LIN {X 0,Y 240.365,Z 392.146,A -85,B 0,C 180,E1 -19575.841,E2 -19575.841} C_VEL
LIN {X 0,Y 237.753,Z 387.976,A -85,B 0,C 180,E1 -19576.695,E2 -19576.695} C_VEL
LIN {X 0,Y 237.227,Z 386.044,A -85,B 0,C 180,E1 -19576.943,E2 -19576.943} C_VEL
LIN {X 0,Y 236.786,Z 383.152,A -85,B 0,C 180,E1 -19580.508,E2 -19580.508} C_VEL
LIN {X 0,Y 236.424,Z 380.849,A -85,B 0,C 180,E1 -19583.522,E2 -19583.522} C_VEL
LIN {X 0,Y 235.914,Z 377.933,A -85,B 0,C 180,E1 -19587.573,E2 -19587.573} C_VEL
LIN {X 0,Y 235.569,Z 375.427,A -85,B 0,C 180,E1 -19591.488,E2 -19591.488} C_VEL
LIN {X 0,Y 235.207,Z 373.215,A -85,B 0,C 180,E1 -19595.272,E2 -19595.272} C_VEL
LIN {X 0,Y 234.997,Z 371.839,A -85,B 0,C 180,E1 -19597.991,E2 -19597.991} C_VEL
LIN {X 0,Y 235.1,Z 371.828,A -85,B 0,C 180,E1 -19603.06,E2 -19603.06} C_VEL
LIN {X 0,Y 235.15,Z 371.825,A -85,B 0,C 180,E1 -19607.924,E2 -19607.924} C_VEL
LIN {X 0,Y 235.394,Z 371.792,A -85,B 0,C 180,E1 -19611.415,E2 -19611.415} C_VEL
LIN {X 0,Y 235.41,Z 371.786,A -85,B 0,C 180,E1 -19613.142,E2 -19613.142} C_VEL
LIN {X 0,Y 235.6,Z 371.764,A -85,B 0,C 180,E1 -19618.291,E2 -19618.291} C_VEL
LIN {X 0,Y 235.6,Z 371.763,A -85,B 0,C 180,E1 -19621.71,E2 -19621.71} C_VEL
LIN {X 0,Y 235.41,Z 371.779,A -85,B 0,C 180,E1 -19626.859,E2 -19626.859} C_VEL
LIN {X 0,Y 235.257,Z 371.795,A -85,B 0,C 180,E1 -19630.326,E2 -19630.326} C_VEL
LIN {X 0,Y 235.117,Z 371.816,A -85,B 0,C 180,E1 -19635.606,E2 -19635.606} C_VEL
LIN {X 0,Y 235.011,Z 371.808,A -85,B 0,C 180,E1 -19639.206,E2 -19639.206} C_VEL
LIN {X 0,Y 234.956,Z 371.835,A -85,B 0,C 180,E1 -19642.884,E2 -19642.884} C_VEL
LIN {X 0,Y 234.97,Z 371.815,A -85,B 0,C 180,E1 -19646.657,E2 -19646.657} C_VEL
LIN {X 0,Y 234.926,Z 371.847,A -85,B 0,C 180,E1 -19650.569,E2 -19650.569} C_VEL
LIN {X 0,Y 234.964,Z 371.826,A -85,B 0,C 180,E1 -19654.633,E2 -19654.633} C_VEL
LIN {X 0,Y 234.945,Z 371.844,A -85,B 0,C 180,E1 -19658.944,E2 -19658.944} C_VEL
LIN {X 0,Y 234.877,Z 371.898,A -85,B 0,C 180,E1 -19662.586,E2 -19662.586} C_VEL
LIN {X 0,Y 235.767,Z 374.534,A -85,B 0,C 180,E1 -19662.962,E2 -19662.962} C_VEL
LIN {X 0,Y 237.695,Z 376.657,A -85,B 0,C 180,E1 -19663.576,E2 -19663.576} C_VEL
LIN {X 0,Y 240.331,Z 380.728,A -85,B 0,C 180,E1 -19664.475,E2 -19664.475} C_VEL
LIN {X 0,Y 244.031,Z 386.932,A -85,B 0,C 180,E1 -19665.775,E2 -19665.775} C_VEL
LIN {X 0,Y 247.642,Z 393.701,A -85,B 0,C 180,E1 -19667.125,E2 -19667.125} C_VEL
LIN {X 0,Y 252.641,Z 405.359,A -85,B 0,C 180,E1 -19669.292,E2 -19669.292} C_VEL
LIN {X 0,Y 256.805,Z 418.111,A -85,B 0,C 180,E1 -19671.571,E2 -19671.571} C_VEL
LIN {X 0,Y 259.553,Z 429.821,A -85,B 0,C 180,E1 -19673.664,E2 -19673.664} C_VEL
LIN {X 0,Y 260.589,Z 437.318,A -85,B 0,C 180,E1 -19675.014,E2 -19675.014} C_VEL
LIN {X 0,Y 257.442,Z 449.414,A -85,B 0,C 180,E1 -19676.673,E2 -19676.673} C_VEL
LIN {X 0,Y 253.705,Z 461.584,A -85,B 0,C 180,E1 -19678.707,E2 -19678.707} C_VEL
LIN {X 0,Y 250.336,Z 471.991,A -85,B 0,C 180,E1 -19680.859,E2 -19680.859} C_VEL
LIN {X 0,Y 246.821,Z 481.962,A -85,B 0,C 180,E1 -19683.354,E2 -19683.354} C_VEL
LIN {X 0,Y 243.43,Z 491.106,A -85,B 0,C 180,E1 -19686.159,E2 -19686.159} C_VEL
LIN {X 0,Y 240.902,Z 497.706,A -85,B 0,C 180,E1 -19688.612,E2 -19688.612} C_VEL
LIN {X 0,Y 238.819,Z 503.332,A -85,B 0,C 180,E1 -19691.112,E2 -19691.112} C_VEL
LIN {X 0,Y 236.494,Z 509.456,A -85,B 0,C 180,E1 -19694.486,E2 -19694.486} C_VEL
LIN {X 0,Y 234.943,Z 514.169,A -85,B 0,C 180,E1 -19697.912,E2 -19697.912} C_VEL
LIN {X 0,Y 233.837,Z 517.618,A -85,B 0,C 180,E1 -19701.356,E2 -19701.356} C_VEL
LIN {X 0,Y 233.305,Z 519.888,A -85,B 0,C 180,E1 -19704.814,E2 -19704.814} C_VEL
LIN {X 0,Y 233.028,Z 521.046,A -85,B 0,C 180,E1 -19708.271,E2 -19708.271} C_VEL
LIN {X 0,Y 233.027,Z 521.058,A -85,B 0,C 180,E1 -19711.728,E2 -19711.728} C_VEL
LIN {X 0,Y 233.304,Z 519.95,A -85,B 0,C 180,E1 -19715.184,E2 -19715.184} C_VEL
LIN {X 0,Y 233.835,Z 517.729,A -85,B 0,C 180,E1 -19718.642,E2 -19718.642} C_VEL
LIN {X 0,Y 234.904,Z 514.324,A -85,B 0,C 180,E1 -19722.088,E2 -19722.088} C_VEL
LIN {X 0,Y 236.445,Z 509.661,A -85,B 0,C 180,E1 -19725.515,E2 -19725.515} C_VEL
LIN {X 0,Y 238.775,Z 503.598,A -85,B 0,C 180,E1 -19728.89,E2 -19728.89} C_VEL
LIN {X 0,Y 241.176,Z 497.014,A -85,B 0,C 180,E1 -19731.81,E2 -19731.81} C_VEL
LIN {X 0,Y 244.227,Z 489.035,A -85,B 0,C 180,E1 -19734.661,E2 -19734.661} C_VEL
LIN {X 0,Y 247.76,Z 479.453,A -85,B 0,C 180,E1 -19737.448,E2 -19737.448} C_VEL
LIN {X 0,Y 251.105,Z 469.547,A -85,B 0,C 180,E1 -19739.814,E2 -19739.814} C_VEL
LIN {X 0,Y 254.873,Z 457.976,A -85,B 0,C 180,E1 -19742.059,E2 -19742.059} C_VEL
LIN {X 0,Y 258.281,Z 446.345,A -85,B 0,C 180,E1 -19743.904,E2 -19743.904} C_VEL
LIN {X 0,Y 260.705,Z 436.623,A -85,B 0,C 180,E1 -19745.22,E2 -19745.22} C_VEL
LIN {X 0,Y 258.709,Z 425.382,A -85,B 0,C 180,E1 -19747.255,E2 -19747.255} C_VEL
LIN {X 0,Y 255.207,Z 412.553,A -85,B 0,C 180,E1 -19749.549,E2 -19749.549} C_VEL
LIN {X 0,Y 250.965,Z 401.064,A -85,B 0,C 180,E1 -19751.64,E2 -19751.64} C_VEL
LIN {X 0,Y 245.554,Z 389.421,A -85,B 0,C 180,E1 -19753.827,E2 -19753.827} C_VEL
LIN {X 0,Y 240.349,Z 380.733,A -85,B 0,C 180,E1 -19755.678,E2 -19755.678} C_VEL
LIN {X 0,Y 238.22,Z 377.466,A -85,B 0,C 180,E1 -19756.408,E2 -19756.408} C_VEL
LIN {X 0,Y 237.051,Z 376.15,A -85,B 0,C 180,E1 -19756.778,E2 -19756.778} C_VEL
LIN {X 0,Y 235.396,Z 373.796,A -85,B 0,C 180,E1 -19757.338,E2 -19757.338} C_VEL
LIN {X 0,Y 234.883,Z 371.853,A -85,B 0,C 180,E1 -19757.607,E2 -19757.607} C_VEL
LIN {X 0,Y 234.953,Z 371.842,A -85,B 0,C 180,E1 -19761.085,E2 -19761.085} C_VEL
LIN {X 0,Y 234.959,Z 371.832,A -85,B 0,C 180,E1 -19765.367,E2 -19765.367} C_VEL
LIN {X 0,Y 234.968,Z 371.841,A -85,B 0,C 180,E1 -19770.157,E2 -19770.157} C_VEL
LIN {X 0,Y 234.992,Z 371.815,A -85,B 0,C 180,E1 -19773.793,E2 -19773.793} C_VEL
LIN {X 0,Y 235.009,Z 371.806,A -85,B 0,C 180,E1 -19778.969,E2 -19778.969} C_VEL
LIN {X 0,Y 235.095,Z 371.825,A -85,B 0,C 180,E1 -19783.059,E2 -19783.059} C_VEL
LIN {X 0,Y 235.117,Z 371.793,A -85,B 0,C 180,E1 -19787.922,E2 -19787.922} C_VEL
LIN {X 0,Y 235.389,Z 371.788,A -85,B 0,C 180,E1 -19791.414,E2 -19791.414} C_VEL
LIN {X 0,Y 235.404,Z 371.788,A -85,B 0,C 180,E1 -19793.141,E2 -19793.141} C_VEL
LIN {X 0,Y 235.595,Z 371.764,A -85,B 0,C 180,E1 -19798.29,E2 -19798.29} C_VEL
LIN {X 0,Y 235.595,Z 371.766,A -85,B 0,C 180,E1 -19801.709,E2 -19801.709} C_VEL
LIN {X 0,Y 235.404,Z 371.788,A -85,B 0,C 180,E1 -19806.858,E2 -19806.858} C_VEL
LIN {X 0,Y 235.251,Z 371.806,A -85,B 0,C 180,E1 -19810.326,E2 -19810.326} C_VEL
LIN {X 0,Y 235.112,Z 371.817,A -85,B 0,C 180,E1 -19815.606,E2 -19815.606} C_VEL
LIN {X 0,Y 235.007,Z 371.836,A -85,B 0,C 180,E1 -19819.206,E2 -19819.206} C_VEL
LIN {X 0,Y 234.991,Z 371.84,A -85,B 0,C 180,E1 -19822.01,E2 -19822.01} C_VEL
LIN {X 0,Y 235.417,Z 374.315,A -85,B 0,C 180,E1 -19826.602,E2 -19826.602} C_VEL
LIN {X 0,Y 235.77,Z 376.689,A -85,B 0,C 180,E1 -19830.447,E2 -19830.447} C_VEL
LIN {X 0,Y 236.166,Z 379.419,A -85,B 0,C 180,E1 -19834.431,E2 -19834.431} C_VEL
LIN {X 0,Y 236.671,Z 382.515,A -85,B 0,C 180,E1 -19838.62,E2 -19838.62} C_VEL
LIN {X 0,Y 237.11,Z 385.372,A -85,B 0,C 180,E1 -19842.184,E2 -19842.184} C_VEL
LIN {X 0,Y 237.201,Z 386.06,A -85,B 0,C 180,E1 -19843.01,E2 -19843.01} C_VEL
LIN {X 0,Y 238.311,Z 389.145,A -85,B 0,C 180,E1 -19843.436,E2 -19843.436} C_VEL
LIN {X 0,Y 240.316,Z 392.138,A -85,B 0,C 180,E1 -19844.08,E2 -19844.08} C_VEL
LIN {X 0,Y 242.022,Z 395.595,A -85,B 0,C 180,E1 -19844.662,E2 -19844.662} C_VEL
LIN {X 0,Y 243.385,Z 398.6,A -85,B 0,C 180,E1 -19845.16,E2 -19845.16} C_VEL
LIN {X 0,Y 244.56,Z 403.788,A -85,B 0,C 180,E1 -19845.767,E2 -19845.767} C_VEL
LIN {X 0,Y 245.066,Z 416.913,A -85,B 0,C 180,E1 -19846.969,E2 -19846.969} C_VEL
LIN {X 0,Y 245.512,Z 422.315,A -85,B 0,C 180,E1 -19847.6,E2 -19847.6} C_VEL
LIN {X 0,Y 245.845,Z 423.998,A -85,B 0,C 180,E1 -19847.847,E2 -19847.847} C_VEL
LIN {X 0,Y 248.348,Z 436.665,A -85,B 0,C 180,E1 -19849.824,E2 -19849.824} C_VEL
LIN {X 0,Y 249.673,Z 447.615,A -85,B 0,C 180,E1 -19851.571,E2 -19851.571} C_VEL
LIN {X 0,Y 250.293,Z 459.212,A -85,B 0,C 180,E1 -19853.528,E2 -19853.528} C_VEL
LIN {X 0,Y 250.148,Z 467.524,A -85,B 0,C 180,E1 -19855,E2 -19855} C_VEL
LIN {X 0,Y 246.211,Z 479.542,A -85,B 0,C 180,E1 -19856.914,E2 -19856.914} C_VEL
LIN {X 0,Y 242.5,Z 490.354,A -85,B 0,C 180,E1 -19859.042,E2 -19859.042} C_VEL
LIN {X 0,Y 238.921,Z 500.373,A -85,B 0,C 180,E1 -19861.446,E2 -19861.446} C_VEL
LIN {X 0,Y 235.371,Z 510.194,A -85,B 0,C 180,E1 -19864.345,E2 -19864.345} C_VEL
LIN {X 0,Y 232.244,Z 518.392,A -85,B 0,C 180,E1 -19867.306,E2 -19867.306} C_VEL
LIN {X 0,Y 229.865,Z 525.192,A -85,B 0,C 180,E1 -19870.348,E2 -19870.348} C_VEL
LIN {X 0,Y 227.851,Z 531.486,A -85,B 0,C 180,E1 -19873.884,E2 -19873.884} C_VEL
LIN {X 0,Y 226.472,Z 536.364,A -85,B 0,C 180,E1 -19877.455,E2 -19877.455} C_VEL
LIN {X 0,Y 225.859,Z 539.958,A -85,B 0,C 180,E1 -19881.05,E2 -19881.05} C_VEL
LIN {X 0,Y 225.762,Z 542.491,A -85,B 0,C 180,E1 -19884.979,E2 -19884.979} C_VEL
LIN {X 0,Y 225.823,Z 543.533,A -85,B 0,C 180,E1 -19888.217,E2 -19888.217} C_VEL
LIN {X 0,Y 225.879,Z 543.692,A -85,B 0,C 180,E1 -19890.001,E2 -19890.001} C_VEL
LIN {X 0,Y 225.738,Z 543.065,A -85,B 0,C 180,E1 -19893.571,E2 -19893.571} C_VEL
LIN {X 0,Y 225.79,Z 541.267,A -85,B 0,C 180,E1 -19897.153,E2 -19897.153} C_VEL
LIN {X 0,Y 226.079,Z 538.274,A -85,B 0,C 180,E1 -19900.75,E2 -19900.75} C_VEL
LIN {X 0,Y 227.108,Z 534.042,A -85,B 0,C 180,E1 -19904.334,E2 -19904.334} C_VEL
LIN {X 0,Y 228.777,Z 528.453,A -85,B 0,C 180,E1 -19907.891,E2 -19907.891} C_VEL
LIN {X 0,Y 231.143,Z 521.361,A -85,B 0,C 180,E1 -19911.4,E2 -19911.4} C_VEL
LIN {X 0,Y 233.997,Z 513.801,A -85,B 0,C 180,E1 -19914.393,E2 -19914.393} C_VEL
LIN {X 0,Y 237.628,Z 503.825,A -85,B 0,C 180,E1 -19917.576,E2 -19917.576} C_VEL
LIN {X 0,Y 241.296,Z 493.766,A -85,B 0,C 180,E1 -19920.161,E2 -19920.161} C_VEL
LIN {X 0,Y 245.546,Z 481.496,A -85,B 0,C 180,E1 -19922.701,E2 -19922.701} C_VEL
LIN {X 0,Y 249.696,Z 468.862,A -85,B 0,C 180,E1 -19924.775,E2 -19924.775} C_VEL
LIN {X 0,Y 250.205,Z 466.104,A -85,B 0,C 180,E1 -19925.212,E2 -19925.212} C_VEL
LIN {X 0,Y 250.129,Z 454.413,A -85,B 0,C 180,E1 -19927.251,E2 -19927.251} C_VEL
LIN {X 0,Y 249.121,Z 442.557,A -85,B 0,C 180,E1 -19929.202,E2 -19929.202} C_VEL
LIN {X 0,Y 247.216,Z 430.307,A -85,B 0,C 180,E1 -19931.117,E2 -19931.117} C_VEL
LIN {X 0,Y 243.831,Z 416.677,A -85,B 0,C 180,E1 -19933.258,E2 -19933.258} C_VEL
LIN {X 0,Y 239.847,Z 404.951,A -85,B 0,C 180,E1 -19935.158,E2 -19935.158} C_VEL
LIN {X 0,Y 237.479,Z 399.928,A -85,B 0,C 180,E1 -19936.083,E2 -19936.083} C_VEL
LIN {X 0,Y 235.391,Z 395.789,A -85,B 0,C 180,E1 -19936.883,E2 -19936.883} C_VEL
LIN {X 0,Y 233.368,Z 392.047,A -85,B 0,C 180,E1 -19937.617,E2 -19937.617} C_VEL
LIN {X 0,Y 232.475,Z 390.688,A -85,B 0,C 180,E1 -19937.927,E2 -19937.927} C_VEL
LIN {X 0,Y 230.569,Z 387.673,A -85,B 0,C 180,E1 -19938.61,E2 -19938.61} C_VEL
LIN {X 0,Y 229.99,Z 385.549,A -85,B 0,C 180,E1 -19938.915,E2 -19938.915} C_VEL
LIN {X 0,Y 229.487,Z 382.624,A -85,B 0,C 180,E1 -19942.774,E2 -19942.774} C_VEL
LIN {X 0,Y 229.09,Z 380.015,A -85,B 0,C 180,E1 -19946.482,E2 -19946.482} C_VEL
LIN {X 0,Y 228.665,Z 377.405,A -85,B 0,C 180,E1 -19950.544,E2 -19950.544} C_VEL
LIN {X 0,Y 228.33,Z 375.085,A -85,B 0,C 180,E1 -19954.474,E2 -19954.474} C_VEL
LIN {X 0,Y 228.007,Z 373.088,A -85,B 0,C 180,E1 -19958.292,E2 -19958.292} C_VEL
LIN {X 0,Y 228.007,Z 372.71,A -85,B 0,C 180,E1 -19962.047,E2 -19962.047} C_VEL
LIN {X 0,Y 228.069,Z 372.705,A -85,B 0,C 180,E1 -19965.728,E2 -19965.728} C_VEL
LIN {X 0,Y 228.329,Z 372.672,A -85,B 0,C 180,E1 -19971.147,E2 -19971.147} C_VEL
LIN {X 0,Y 228.362,Z 372.665,A -85,B 0,C 180,E1 -19972.929,E2 -19972.929} C_VEL
LIN {X 0,Y 228.559,Z 372.642,A -85,B 0,C 180,E1 -19978.238,E2 -19978.238} C_VEL
LIN {X 0,Y 228.559,Z 372.64,A -85,B 0,C 180,E1 -19981.762,E2 -19981.762} C_VEL
LIN {X 0,Y 228.362,Z 372.657,A -85,B 0,C 180,E1 -19987.071,E2 -19987.071} C_VEL
LIN {X 0,Y 228.171,Z 372.67,A -85,B 0,C 180,E1 -19990.65,E2 -19990.65} C_VEL
LIN {X 0,Y 228.068,Z 372.671,A -85,B 0,C 180,E1 -19994.272,E2 -19994.272} C_VEL
LIN {X 0,Y 228.006,Z 372.699,A -85,B 0,C 180,E1 -19997.953,E2 -19997.953} C_VEL
LIN {X 0,Y 227.92,Z 372.7,A -85,B 0,C 180,E1 -20002.321,E2 -20002.321} C_VEL
LIN {X 0,Y 227.945,Z 372.689,A -85,B 0,C 180,E1 -20006.602,E2 -20006.602} C_VEL
LIN {X 0,Y 227.901,Z 372.722,A -85,B 0,C 180,E1 -20010.291,E2 -20010.291} C_VEL
LIN {X 0,Y 227.893,Z 372.7,A -85,B 0,C 180,E1 -20013.718,E2 -20013.718} C_VEL
LIN {X 0,Y 227.873,Z 372.726,A -85,B 0,C 180,E1 -20018.086,E2 -20018.086} C_VEL
LIN {X 0,Y 227.84,Z 372.737,A -85,B 0,C 180,E1 -20020.64,E2 -20020.64} C_VEL
LIN {X 0,Y 228.705,Z 375.293,A -85,B 0,C 180,E1 -20021.039,E2 -20021.039} C_VEL
LIN {X 0,Y 230.755,Z 377.617,A -85,B 0,C 180,E1 -20021.757,E2 -20021.757} C_VEL
LIN {X 0,Y 233.487,Z 381.79,A -85,B 0,C 180,E1 -20022.776,E2 -20022.776} C_VEL
LIN {X 0,Y 234.607,Z 383.303,A -85,B 0,C 180,E1 -20023.182,E2 -20023.182} C_VEL
LIN {X 0,Y 237.64,Z 388.184,A -85,B 0,C 180,E1 -20024.322,E2 -20024.322} C_VEL
LIN {X 0,Y 242.189,Z 396.617,A -85,B 0,C 180,E1 -20026.156,E2 -20026.156} C_VEL
LIN {X 0,Y 246.882,Z 407.826,A -85,B 0,C 180,E1 -20028.354,E2 -20028.354} C_VEL
LIN {X 0,Y 250.522,Z 419.001,A -85,B 0,C 180,E1 -20030.486,E2 -20030.486} C_VEL
LIN {X 0,Y 253.168,Z 430.055,A -85,B 0,C 180,E1 -20032.567,E2 -20032.567} C_VEL
LIN {X 0,Y 254.483,Z 438.888,A -85,B 0,C 180,E1 -20034.255,E2 -20034.255} C_VEL
LIN {X 0,Y 251.197,Z 450.93,A -85,B 0,C 180,E1 -20035.974,E2 -20035.974} C_VEL
LIN {X 0,Y 247.655,Z 461.936,A -85,B 0,C 180,E1 -20037.852,E2 -20037.852} C_VEL
LIN {X 0,Y 244.059,Z 472.582,A -85,B 0,C 180,E1 -20040.099,E2 -20040.099} C_VEL
LIN {X 0,Y 240.456,Z 482.315,A -85,B 0,C 180,E1 -20042.59,E2 -20042.59} C_VEL
LIN {X 0,Y 236.933,Z 491.457,A -85,B 0,C 180,E1 -20045.463,E2 -20045.463} C_VEL
LIN {X 0,Y 234.286,Z 498.057,A -85,B 0,C 180,E1 -20047.977,E2 -20047.977} C_VEL
LIN {X 0,Y 232.082,Z 503.683,A -85,B 0,C 180,E1 -20050.542,E2 -20050.542} C_VEL
LIN {X 0,Y 230.228,Z 508.403,A -85,B 0,C 180,E1 -20053.141,E2 -20053.141} C_VEL
LIN {X 0,Y 228.342,Z 513.477,A -85,B 0,C 180,E1 -20056.653,E2 -20056.653} C_VEL
LIN {X 0,Y 227.331,Z 516.395,A -85,B 0,C 180,E1 -20059.309,E2 -20059.309} C_VEL
LIN {X 0,Y 226.382,Z 519.591,A -85,B 0,C 180,E1 -20063.433,E2 -20063.433} C_VEL
LIN {X 0,Y 226.111,Z 520.949,A -85,B 0,C 180,E1 -20066.435,E2 -20066.435} C_VEL
LIN {X 0,Y 225.919,Z 521.547,A -85,B 0,C 180,E1 -20069.999,E2 -20069.999} C_VEL
LIN {X 0,Y 226.088,Z 520.987,A -85,B 0,C 180,E1 -20073.564,E2 -20073.564} C_VEL
LIN {X 0,Y 226.491,Z 519.329,A -85,B 0,C 180,E1 -20077.129,E2 -20077.129} C_VEL
LIN {X 0,Y 227.318,Z 516.526,A -85,B 0,C 180,E1 -20080.69,E2 -20080.69} C_VEL
LIN {X 0,Y 228.716,Z 512.504,A -85,B 0,C 180,E1 -20084.23,E2 -20084.23} C_VEL
LIN {X 0,Y 230.799,Z 507.158,A -85,B 0,C 180,E1 -20087.728,E2 -20087.728} C_VEL
LIN {X 0,Y 233.367,Z 500.345,A -85,B 0,C 180,E1 -20091.185,E2 -20091.185} C_VEL
LIN {X 0,Y 236.849,Z 491.814,A -85,B 0,C 180,E1 -20094.545,E2 -20094.545} C_VEL
LIN {X 0,Y 240.344,Z 482.74,A -85,B 0,C 180,E1 -20097.422,E2 -20097.422} C_VEL
LIN {X 0,Y 243.753,Z 473.62,A -85,B 0,C 180,E1 -20099.785,E2 -20099.785} C_VEL
LIN {X 0,Y 247.51,Z 462.49,A -85,B 0,C 180,E1 -20102.167,E2 -20102.167} C_VEL
LIN {X 0,Y 251.417,Z 450.423,A -85,B 0,C 180,E1 -20104.232,E2 -20104.232} C_VEL
LIN {X 0,Y 254.499,Z 439.294,A -85,B 0,C 180,E1 -20105.809,E2 -20105.809} C_VEL
LIN {X 0,Y 253.158,Z 429.641,A -85,B 0,C 180,E1 -20107.643,E2 -20107.643} C_VEL
LIN {X 0,Y 250.331,Z 418.167,A -85,B 0,C 180,E1 -20109.808,E2 -20109.808} C_VEL
LIN {X 0,Y 246.696,Z 407.16,A -85,B 0,C 180,E1 -20111.904,E2 -20111.904} C_VEL
LIN {X 0,Y 241.928,Z 395.995,A -85,B 0,C 180,E1 -20114.117,E2 -20114.117} C_VEL
LIN {X 0,Y 237.89,Z 388.617,A -85,B 0,C 180,E1 -20115.737,E2 -20115.737} C_VEL
LIN {X 0,Y 236.099,Z 385.655,A -85,B 0,C 180,E1 -20116.425,E2 -20116.425} C_VEL
LIN {X 0,Y 233.646,Z 381.958,A -85,B 0,C 180,E1 -20117.333,E2 -20117.333} C_VEL
LIN {X 0,Y 231.567,Z 378.932,A -85,B 0,C 180,E1 -20118.11,E2 -20118.11} C_VEL
LIN {X 0,Y 230.784,Z 377.645,A -85,B 0,C 180,E1 -20118.401,E2 -20118.401} C_VEL
LIN {X 0,Y 228.634,Z 375.23,A -85,B 0,C 180,E1 -20119.157,E2 -20119.157} C_VEL
LIN {X 0,Y 227.853,Z 372.728,A -85,B 0,C 180,E1 -20119.575,E2 -20119.575} C_VEL
LIN {X 0,Y 227.899,Z 372.724,A -85,B 0,C 180,E1 -20124.131,E2 -20124.131} C_VEL
LIN {X 0,Y 227.871,Z 372.712,A -85,B 0,C 180,E1 -20128.378,E2 -20128.378} C_VEL
LIN {X 0,Y 227.884,Z 372.698,A -85,B 0,C 180,E1 -20132.445,E2 -20132.445} C_VEL
LIN {X 0,Y 227.913,Z 372.719,A -85,B 0,C 180,E1 -20136.367,E2 -20136.367} C_VEL
LIN {X 0,Y 227.941,Z 372.686,A -85,B 0,C 180,E1 -20140.174,E2 -20140.174} C_VEL
LIN {X 0,Y 228.056,Z 372.7,A -85,B 0,C 180,E1 -20143.898,E2 -20143.898} C_VEL
LIN {X 0,Y 228.074,Z 372.667,A -85,B 0,C 180,E1 -20147.543,E2 -20147.543} C_VEL
LIN {X 0,Y 228.323,Z 372.669,A -85,B 0,C 180,E1 -20151.147,E2 -20151.147} C_VEL
LIN {X 0,Y 228.357,Z 372.667,A -85,B 0,C 180,E1 -20152.928,E2 -20152.928} C_VEL
LIN {X 0,Y 228.553,Z 372.641,A -85,B 0,C 180,E1 -20158.238,E2 -20158.238} C_VEL
LIN {X 0,Y 228.554,Z 372.643,A -85,B 0,C 180,E1 -20161.762,E2 -20161.762} C_VEL
LIN {X 0,Y 228.356,Z 372.667,A -85,B 0,C 180,E1 -20167.071,E2 -20167.071} C_VEL
LIN {X 0,Y 228.165,Z 372.69,A -85,B 0,C 180,E1 -20170.65,E2 -20170.65} C_VEL
LIN {X 0,Y 228.063,Z 372.701,A -85,B 0,C 180,E1 -20174.272,E2 -20174.272} C_VEL
LIN {X 0,Y 228.001,Z 372.705,A -85,B 0,C 180,E1 -20177.953,E2 -20177.953} C_VEL
LIN {X 0,Y 227.94,Z 372.717,A -85,B 0,C 180,E1 -20179.825,E2 -20179.825} C_VEL
LIN {X 0,Y 228.07,Z 373.495,A -85,B 0,C 180,E1 -20182.416,E2 -20182.416} C_VEL
LIN {X 0,Y 228.466,Z 375.895,A -85,B 0,C 180,E1 -20186.865,E2 -20186.865} C_VEL
LIN {X 0,Y 228.85,Z 378.715,A -85,B 0,C 180,E1 -20191.471,E2 -20191.471} C_VEL
LIN {X 0,Y 229.289,Z 381.526,A -85,B 0,C 180,E1 -20195.617,E2 -20195.617} C_VEL
LIN {X 0,Y 229.933,Z 385.158,A -85,B 0,C 180,E1 -20200.53,E2 -20200.53} C_VEL
LIN {X 0,Y 229.974,Z 385.548,A -85,B 0,C 180,E1 -20201.019,E2 -20201.019} C_VEL
LIN {X 0,Y 231.049,Z 388.684,A -85,B 0,C 180,E1 -20201.501,E2 -20201.501} C_VEL
LIN {X 0,Y 233.27,Z 391.819,A -85,B 0,C 180,E1 -20202.272,E2 -20202.272} C_VEL
LIN {X 0,Y 235.336,Z 395.727,A -85,B 0,C 180,E1 -20203.028,E2 -20203.028} C_VEL
LIN {X 0,Y 236.747,Z 398.488,A -85,B 0,C 180,E1 -20203.572,E2 -20203.572} C_VEL
LIN {X 0,Y 239.144,Z 403.362,A -85,B 0,C 180,E1 -20204.485,E2 -20204.485} C_VEL
LIN {X 0,Y 241.953,Z 410.536,A -85,B 0,C 180,E1 -20205.708,E2 -20205.708} C_VEL
LIN {X 0,Y 245.208,Z 421.548,A -85,B 0,C 180,E1 -20207.458,E2 -20207.458} C_VEL
LIN {X 0,Y 245.845,Z 423.998,A -85,B 0,C 180,E1 -20207.847,E2 -20207.847} C_VEL
LIN {X 0,Y 246.467,Z 429.079,A -85,B 0,C 180,E1 -20208.532,E2 -20208.532} C_VEL
LIN {X 0,Y 246.138,Z 434.527,A -85,B 0,C 180,E1 -20209.122,E2 -20209.122} C_VEL
LIN {X 0,Y 244.334,Z 445.278,A -85,B 0,C 180,E1 -20210.273,E2 -20210.273} C_VEL
LIN {X 0,Y 243.794,Z 450.476,A -85,B 0,C 180,E1 -20210.973,E2 -20210.973} C_VEL
LIN {X 0,Y 243.798,Z 452.076,A -85,B 0,C 180,E1 -20211.239,E2 -20211.239} C_VEL
LIN {X 0,Y 244.081,Z 463.437,A -85,B 0,C 180,E1 -20213.275,E2 -20213.275} C_VEL
LIN {X 0,Y 243.907,Z 468.567,A -85,B 0,C 180,E1 -20214.24,E2 -20214.24} C_VEL
LIN {X 0,Y 239.54,Z 481.348,A -85,B 0,C 180,E1 -20216.374,E2 -20216.374} C_VEL
LIN {X 0,Y 235.086,Z 493.575,A -85,B 0,C 180,E1 -20218.957,E2 -20218.957} C_VEL
LIN {X 0,Y 231.044,Z 504.241,A -85,B 0,C 180,E1 -20221.787,E2 -20221.787} C_VEL
LIN {X 0,Y 227.513,Z 513.563,A -85,B 0,C 180,E1 -20224.866,E2 -20224.866} C_VEL
LIN {X 0,Y 224.458,Z 521.11,A -85,B 0,C 180,E1 -20227.931,E2 -20227.931} C_VEL
LIN {X 0,Y 221.94,Z 528.174,A -85,B 0,C 180,E1 -20231.54,E2 -20231.54} C_VEL
LIN {X 0,Y 220.135,Z 533.742,A -85,B 0,C 180,E1 -20235.203,E2 -20235.203} C_VEL
LIN {X 0,Y 219.058,Z 537.967,A -85,B 0,C 180,E1 -20238.902,E2 -20238.902} C_VEL
LIN {X 0,Y 218.625,Z 540.943,A -85,B 0,C 180,E1 -20242.613,E2 -20242.613} C_VEL
LIN {X 0,Y 218.641,Z 542.729,A -85,B 0,C 180,E1 -20246.315,E2 -20246.315} C_VEL
LIN {X 0,Y 218.81,Z 543.346,A -85,B 0,C 180,E1 -20250.001,E2 -20250.001} C_VEL
LIN {X 0,Y 218.647,Z 542.716,A -85,B 0,C 180,E1 -20253.687,E2 -20253.687} C_VEL
LIN {X 0,Y 218.69,Z 540.916,A -85,B 0,C 180,E1 -20257.386,E2 -20257.386} C_VEL
LIN {X 0,Y 219.059,Z 537.923,A -85,B 0,C 180,E1 -20261.099,E2 -20261.099} C_VEL
LIN {X 0,Y 220.152,Z 533.689,A -85,B 0,C 180,E1 -20264.797,E2 -20264.797} C_VEL
LIN {X 0,Y 221.941,Z 528.099,A -85,B 0,C 180,E1 -20268.462,E2 -20268.462} C_VEL
LIN {X 0,Y 224.458,Z 521.007,A -85,B 0,C 180,E1 -20272.07,E2 -20272.07} C_VEL
LIN {X 0,Y 227.486,Z 513.448,A -85,B 0,C 180,E1 -20275.138,E2 -20275.138} C_VEL
LIN {X 0,Y 231.164,Z 503.815,A -85,B 0,C 180,E1 -20278.3,E2 -20278.3} C_VEL
LIN {X 0,Y 235.133,Z 493.413,A -85,B 0,C 180,E1 -20281.038,E2 -20281.038} C_VEL
LIN {X 0,Y 239.544,Z 481.142,A -85,B 0,C 180,E1 -20283.627,E2 -20283.627} C_VEL
LIN {X 0,Y 243.856,Z 468.502,A -85,B 0,C 180,E1 -20285.734,E2 -20285.734} C_VEL
LIN {X 0,Y 243.999,Z 455.668,A -85,B 0,C 180,E1 -20288.086,E2 -20288.086} C_VEL
LIN {X 0,Y 242.91,Z 441.93,A -85,B 0,C 180,E1 -20290.442,E2 -20290.442} C_VEL
LIN {X 0,Y 241.157,Z 430.791,A -85,B 0,C 180,E1 -20292.276,E2 -20292.276} C_VEL
LIN {X 0,Y 237.893,Z 417.634,A -85,B 0,C 180,E1 -20294.488,E2 -20294.488} C_VEL
LIN {X 0,Y 234.926,Z 408.704,A -85,B 0,C 180,E1 -20296.035,E2 -20296.035} C_VEL
LIN {X 0,Y 231.654,Z 401.363,A -85,B 0,C 180,E1 -20297.47,E2 -20297.47} C_VEL
LIN {X 0,Y 228.463,Z 395.691,A -85,B 0,C 180,E1 -20298.741,E2 -20298.741} C_VEL
LIN {X 0,Y 226.406,Z 392,A -85,B 0,C 180,E1 -20299.557,E2 -20299.557} C_VEL
LIN {X 0,Y 225.713,Z 390.621,A -85,B 0,C 180,E1 -20299.839,E2 -20299.839} C_VEL
LIN {X 0,Y 223.485,Z 387.605,A -85,B 0,C 180,E1 -20300.686,E2 -20300.686} C_VEL
LIN {X 0,Y 222.657,Z 385.012,A -85,B 0,C 180,E1 -20301.136,E2 -20301.136} C_VEL
LIN {X 0,Y 222.195,Z 382.085,A -85,B 0,C 180,E1 -20305.325,E2 -20305.325} C_VEL
LIN {X 0,Y 221.774,Z 379.363,A -85,B 0,C 180,E1 -20309.534,E2 -20309.534} C_VEL
LIN {X 0,Y 221.45,Z 376.969,A -85,B 0,C 180,E1 -20313.621,E2 -20313.621} C_VEL
LIN {X 0,Y 221.098,Z 374.921,A -85,B 0,C 180,E1 -20317.577,E2 -20317.577} C_VEL
LIN {X 0,Y 220.935,Z 373.999,A -85,B 0,C 180,E1 -20319.518,E2 -20319.518} C_VEL
LIN {X 0,Y 220.988,Z 373.586,A -85,B 0,C 180,E1 -20322.571,E2 -20322.571} C_VEL
LIN {X 0,Y 221.03,Z 373.583,A -85,B 0,C 180,E1 -20327.14,E2 -20327.14} C_VEL
LIN {X 0,Y 221.262,Z 373.554,A -85,B 0,C 180,E1 -20330.862,E2 -20330.862} C_VEL
LIN {X 0,Y 221.315,Z 373.545,A -85,B 0,C 180,E1 -20332.703,E2 -20332.703} C_VEL
LIN {X 0,Y 221.517,Z 373.519,A -85,B 0,C 180,E1 -20338.182,E2 -20338.182} C_VEL
LIN {X 0,Y 221.517,Z 373.517,A -85,B 0,C 180,E1 -20341.818,E2 -20341.818} C_VEL
LIN {X 0,Y 221.315,Z 373.535,A -85,B 0,C 180,E1 -20347.298,E2 -20347.298} C_VEL
LIN {X 0,Y 221.115,Z 373.541,A -85,B 0,C 180,E1 -20350.994,E2 -20350.994} C_VEL
LIN {X 0,Y 221.02,Z 373.579,A -85,B 0,C 180,E1 -20356.63,E2 -20356.63} C_VEL
LIN {X 0,Y 220.888,Z 373.559,A -85,B 0,C 180,E1 -20360.487,E2 -20360.487} C_VEL
LIN {X 0,Y 220.866,Z 373.596,A -85,B 0,C 180,E1 -20364.435,E2 -20364.435} C_VEL
LIN {X 0,Y 220.83,Z 373.579,A -85,B 0,C 180,E1 -20368.515,E2 -20368.515} C_VEL
LIN {X 0,Y 220.826,Z 373.581,A -85,B 0,C 180,E1 -20372.755,E2 -20372.755} C_VEL
LIN {X 0,Y 220.842,Z 373.602,A -85,B 0,C 180,E1 -20377.288,E2 -20377.288} C_VEL
LIN {X 0,Y 220.847,Z 373.684,A -85,B 0,C 180,E1 -20378.501,E2 -20378.501} C_VEL
LIN {X 0,Y 221.651,Z 376.192,A -85,B 0,C 180,E1 -20378.918,E2 -20378.918} C_VEL
LIN {X 0,Y 223.631,Z 378.416,A -85,B 0,C 180,E1 -20379.683,E2 -20379.683} C_VEL
LIN {X 0,Y 224.483,Z 379.429,A -85,B 0,C 180,E1 -20380.008,E2 -20380.008} C_VEL
LIN {X 0,Y 226.542,Z 382.669,A -85,B 0,C 180,E1 -20380.868,E2 -20380.868} C_VEL
LIN {X 0,Y 227.861,Z 384.392,A -85,B 0,C 180,E1 -20381.386,E2 -20381.386} C_VEL
LIN {X 0,Y 231.25,Z 389.629,A -85,B 0,C 180,E1 -20382.763,E2 -20382.763} C_VEL
LIN {X 0,Y 234.891,Z 395.831,A -85,B 0,C 180,E1 -20384.288,E2 -20384.288} C_VEL
LIN {X 0,Y 239.012,Z 404.711,A -85,B 0,C 180,E1 -20386.239,E2 -20386.239} C_VEL
LIN {X 0,Y 243.335,Z 416.6,A -85,B 0,C 180,E1 -20388.671,E2 -20388.671} C_VEL
LIN {X 0,Y 246.184,Z 427.476,A -85,B 0,C 180,E1 -20390.844,E2 -20390.844} C_VEL
LIN {X 0,Y 248.118,Z 438.211,A -85,B 0,C 180,E1 -20392.996,E2 -20392.996} C_VEL
LIN {X 0,Y 248.271,Z 440.971,A -85,B 0,C 180,E1 -20393.525,E2 -20393.525} C_VEL
LIN {X 0,Y 244.601,Z 453.612,A -85,B 0,C 180,E1 -20395.425,E2 -20395.425} C_VEL
LIN {X 0,Y 240.989,Z 464.223,A -85,B 0,C 180,E1 -20397.348,E2 -20397.348} C_VEL
LIN {X 0,Y 237.755,Z 473.397,A -85,B 0,C 180,E1 -20399.352,E2 -20399.352} C_VEL
LIN {X 0,Y 233.638,Z 484.104,A -85,B 0,C 180,E1 -20402.208,E2 -20402.208} C_VEL
LIN {X 0,Y 229.99,Z 493.017,A -85,B 0,C 180,E1 -20405.154,E2 -20405.154} C_VEL
LIN {X 0,Y 226.491,Z 501.284,A -85,B 0,C 180,E1 -20408.576,E2 -20408.576} C_VEL
LIN {X 0,Y 224.099,Z 507.275,A -85,B 0,C 180,E1 -20411.722,E2 -20411.722} C_VEL
LIN {X 0,Y 221.867,Z 512.678,A -85,B 0,C 180,E1 -20415.32,E2 -20415.32} C_VEL
LIN {X 0,Y 220.345,Z 516.744,A -85,B 0,C 180,E1 -20418.966,E2 -20418.966} C_VEL
LIN {X 0,Y 219.435,Z 519.592,A -85,B 0,C 180,E1 -20422.639,E2 -20422.639} C_VEL
LIN {X 0,Y 219.031,Z 521.297,A -85,B 0,C 180,E1 -20426.32,E2 -20426.32} C_VEL
LIN {X 0,Y 218.85,Z 521.894,A -85,B 0,C 180,E1 -20429.999,E2 -20429.999} C_VEL
LIN {X 0,Y 219.009,Z 521.334,A -85,B 0,C 180,E1 -20433.679,E2 -20433.679} C_VEL
LIN {X 0,Y 219.434,Z 519.677,A -85,B 0,C 180,E1 -20437.36,E2 -20437.36} C_VEL
LIN {X 0,Y 220.33,Z 516.874,A -85,B 0,C 180,E1 -20441.033,E2 -20441.033} C_VEL
LIN {X 0,Y 221.811,Z 512.852,A -85,B 0,C 180,E1 -20444.683,E2 -20444.683} C_VEL
LIN {X 0,Y 224.012,Z 507.506,A -85,B 0,C 180,E1 -20448.283,E2 -20448.283} C_VEL
LIN {X 0,Y 226.74,Z 500.692,A -85,B 0,C 180,E1 -20451.835,E2 -20451.835} C_VEL
LIN {X 0,Y 230.386,Z 492.161,A -85,B 0,C 180,E1 -20455.281,E2 -20455.281} C_VEL
LIN {X 0,Y 234.057,Z 483.086,A -85,B 0,C 180,E1 -20458.223,E2 -20458.223} C_VEL
LIN {X 0,Y 237.988,Z 472.859,A -85,B 0,C 180,E1 -20460.906,E2 -20460.906} C_VEL
LIN {X 0,Y 241.886,Z 461.847,A -85,B 0,C 180,E1 -20463.257,E2 -20463.257} C_VEL
LIN {X 0,Y 245.915,Z 449.588,A -85,B 0,C 180,E1 -20465.36,E2 -20465.36} C_VEL
LIN {X 0,Y 248.428,Z 440.948,A -85,B 0,C 180,E1 -20466.592,E2 -20466.592} C_VEL
LIN {X 0,Y 246.83,Z 430.03,A -85,B 0,C 180,E1 -20468.785,E2 -20468.785} C_VEL
LIN {X 0,Y 243.968,Z 418.528,A -85,B 0,C 180,E1 -20471.071,E2 -20471.071} C_VEL
LIN {X 0,Y 239.982,Z 406.96,A -85,B 0,C 180,E1 -20473.431,E2 -20473.431} C_VEL
LIN {X 0,Y 236.044,Z 398.094,A -85,B 0,C 180,E1 -20475.347,E2 -20475.347} C_VEL
LIN {X 0,Y 232.097,Z 390.945,A -85,B 0,C 180,E1 -20477.054,E2 -20477.054} C_VEL
LIN {X 0,Y 229.558,Z 387.025,A -85,B 0,C 180,E1 -20478.103,E2 -20478.103} C_VEL
LIN {X 0,Y 226.842,Z 382.97,A -85,B 0,C 180,E1 -20479.192,E2 -20479.192} C_VEL
LIN {X 0,Y 224.751,Z 380.006,A -85,B 0,C 180,E1 -20480.05,E2 -20480.05} C_VEL
LIN {X 0,Y 223.941,Z 378.656,A -85,B 0,C 180,E1 -20480.383,E2 -20480.383} C_VEL
LIN {X 0,Y 221.819,Z 376.486,A -85,B 0,C 180,E1 -20481.19,E2 -20481.19} C_VEL
LIN {X 0,Y 220.885,Z 373.95,A -85,B 0,C 180,E1 -20481.653,E2 -20481.653} C_VEL
LIN {X 0,Y 220.841,Z 373.601,A -85,B 0,C 180,E1 -20481.789,E2 -20481.789} C_VEL
LIN {X 0,Y 220.819,Z 373.587,A -85,B 0,C 180,E1 -20485.841,E2 -20485.841} C_VEL
LIN {X 0,Y 220.867,Z 373.598,A -85,B 0,C 180,E1 -20489.394,E2 -20489.394} C_VEL
LIN {X 0,Y 220.894,Z 373.569,A -85,B 0,C 180,E1 -20493.549,E2 -20493.549} C_VEL
LIN {X 0,Y 220.876,Z 373.581,A -85,B 0,C 180,E1 -20497.553,E2 -20497.553} C_VEL
LIN {X 0,Y 220.983,Z 373.581,A -85,B 0,C 180,E1 -20502.571,E2 -20502.571} C_VEL
LIN {X 0,Y 221.012,Z 373.544,A -85,B 0,C 180,E1 -20507.138,E2 -20507.138} C_VEL
LIN {X 0,Y 221.257,Z 373.551,A -85,B 0,C 180,E1 -20510.861,E2 -20510.861} C_VEL
LIN {X 0,Y 221.31,Z 373.544,A -85,B 0,C 180,E1 -20512.702,E2 -20512.702} C_VEL
LIN {X 0,Y 221.511,Z 373.518,A -85,B 0,C 180,E1 -20518.182,E2 -20518.182} C_VEL
LIN {X 0,Y 221.512,Z 373.52,A -85,B 0,C 180,E1 -20521.818,E2 -20521.818} C_VEL
LIN {X 0,Y 221.309,Z 373.545,A -85,B 0,C 180,E1 -20527.298,E2 -20527.298} C_VEL
LIN {X 0,Y 221.109,Z 373.569,A -85,B 0,C 180,E1 -20530.994,E2 -20530.994} C_VEL
LIN {X 0,Y 221.014,Z 373.577,A -85,B 0,C 180,E1 -20536.63,E2 -20536.63} C_VEL
LIN {X 0,Y 220.92,Z 373.586,A -85,B 0,C 180,E1 -20538.549,E2 -20538.549} C_VEL
LIN {X 0,Y 220.938,Z 374.054,A -85,B 0,C 180,E1 -20540.481,E2 -20540.481} C_VEL
LIN {X 0,Y 221.242,Z 375.965,A -85,B 0,C 180,E1 -20544.391,E2 -20544.391} C_VEL
LIN {X 0,Y 221.594,Z 378.19,A -85,B 0,C 180,E1 -20548.407,E2 -20548.407} C_VEL
LIN {X 0,Y 221.979,Z 380.731,A -85,B 0,C 180,E1 -20552.563,E2 -20552.563} C_VEL
LIN {X 0,Y 222.447,Z 383.653,A -85,B 0,C 180,E1 -20556.89,E2 -20556.89} C_VEL
LIN {X 0,Y 222.641,Z 385.031,A -85,B 0,C 180,E1 -20558.821,E2 -20558.821} C_VEL
LIN {X 0,Y 223.863,Z 388.314,A -85,B 0,C 180,E1 -20559.385,E2 -20559.385} C_VEL
LIN {X 0,Y 226.253,Z 391.564,A -85,B 0,C 180,E1 -20560.292,E2 -20560.292} C_VEL
LIN {X 0,Y 228.231,Z 395.342,A -85,B 0,C 180,E1 -20561.09,E2 -20561.09} C_VEL
LIN {X 0,Y 229.534,Z 397.48,A -85,B 0,C 180,E1 -20561.608,E2 -20561.608} C_VEL
LIN {X 0,Y 232.985,Z 404.32,A -85,B 0,C 180,E1 -20563.038,E2 -20563.038} C_VEL
LIN {X 0,Y 235.741,Z 410.712,A -85,B 0,C 180,E1 -20564.268,E2 -20564.268} C_VEL
LIN {X 0,Y 238.895,Z 420.805,A -85,B 0,C 180,E1 -20566.016,E2 -20566.016} C_VEL
LIN {X 0,Y 241.739,Z 433.58,A -85,B 0,C 180,E1 -20568.127,E2 -20568.127} C_VEL
LIN {X 0,Y 243.382,Z 445.516,A -85,B 0,C 180,E1 -20570.131,E2 -20570.131} C_VEL
LIN {X 0,Y 243.798,Z 452.076,A -85,B 0,C 180,E1 -20571.239,E2 -20571.239} C_VEL
LIN {X 0,Y 243.333,Z 457.097,A -85,B 0,C 180,E1 -20572.001,E2 -20572.001} C_VEL
LIN {X 0,Y 241.88,Z 462.132,A -85,B 0,C 180,E1 -20572.659,E2 -20572.659} C_VEL
LIN {X 0,Y 237.408,Z 472.066,A -85,B 0,C 180,E1 -20573.94,E2 -20573.94} C_VEL
LIN {X 0,Y 234.584,Z 478.43,A -85,B 0,C 180,E1 -20574.94,E2 -20574.94} C_VEL
LIN {X 0,Y 230.348,Z 489.659,A -85,B 0,C 180,E1 -20577.211,E2 -20577.211} C_VEL
LIN {X 0,Y 226.404,Z 499.674,A -85,B 0,C 180,E1 -20579.707,E2 -20579.707} C_VEL
LIN {X 0,Y 222.464,Z 509.491,A -85,B 0,C 180,E1 -20582.738,E2 -20582.738} C_VEL
LIN {X 0,Y 219.095,Z 517.693,A -85,B 0,C 180,E1 -20585.86,E2 -20585.86} C_VEL
LIN {X 0,Y 216.372,Z 524.49,A -85,B 0,C 180,E1 -20589.067,E2 -20589.067} C_VEL
LIN {X 0,Y 214.069,Z 530.783,A -85,B 0,C 180,E1 -20592.815,E2 -20592.815} C_VEL
LIN {X 0,Y 212.526,Z 535.664,A -85,B 0,C 180,E1 -20596.617,E2 -20596.617} C_VEL
LIN {X 0,Y 211.735,Z 539.258,A -85,B 0,C 180,E1 -20600.448,E2 -20600.448} C_VEL
LIN {X 0,Y 211.555,Z 541.636,A -85,B 0,C 180,E1 -20604.281,E2 -20604.281} C_VEL
LIN {X 0,Y 211.641,Z 542.838,A -85,B 0,C 180,E1 -20608.098,E2 -20608.098} C_VEL
LIN {X 0,Y 211.742,Z 542.999,A -85,B 0,C 180,E1 -20610.001,E2 -20610.001} C_VEL
LIN {X 0,Y 211.561,Z 542.368,A -85,B 0,C 180,E1 -20613.81,E2 -20613.81} C_VEL
LIN {X 0,Y 211.608,Z 540.565,A -85,B 0,C 180,E1 -20617.635,E2 -20617.635} C_VEL
LIN {X 0,Y 212.036,Z 537.572,A -85,B 0,C 180,E1 -20621.472,E2 -20621.472} C_VEL
LIN {X 0,Y 213.202,Z 533.335,A -85,B 0,C 180,E1 -20625.291,E2 -20625.291} C_VEL
LIN {X 0,Y 215.121,Z 527.745,A -85,B 0,C 180,E1 -20629.069,E2 -20629.069} C_VEL
LIN {X 0,Y 217.824,Z 520.654,A -85,B 0,C 180,E1 -20632.78,E2 -20632.78} C_VEL
LIN {X 0,Y 221.498,Z 511.861,A -85,B 0,C 180,E1 -20636.374,E2 -20636.374} C_VEL
LIN {X 0,Y 225.253,Z 502.429,A -85,B 0,C 180,E1 -20639.467,E2 -20639.467} C_VEL
LIN {X 0,Y 229.002,Z 493.058,A -85,B 0,C 180,E1 -20641.966,E2 -20641.966} C_VEL
LIN {X 0,Y 233.596,Z 480.786,A -85,B 0,C 180,E1 -20644.603,E2 -20644.603} C_VEL
LIN {X 0,Y 237.615,Z 469.5,A -85,B 0,C 180,E1 -20646.537,E2 -20646.537} C_VEL
LIN {X 0,Y 237.902,Z 457.721,A -85,B 0,C 180,E1 -20648.793,E2 -20648.793} C_VEL
LIN {X 0,Y 237.126,Z 444.861,A -85,B 0,C 180,E1 -20651.124,E2 -20651.124} C_VEL
LIN {X 0,Y 235.648,Z 433.879,A -85,B 0,C 180,E1 -20653.057,E2 -20653.057} C_VEL
LIN {X 0,Y 233.065,Z 422.373,A -85,B 0,C 180,E1 -20655.09,E2 -20655.09} C_VEL
LIN {X 0,Y 230.334,Z 413.205,A -85,B 0,C 180,E1 -20656.765,E2 -20656.765} C_VEL
LIN {X 0,Y 227.053,Z 405.669,A -85,B 0,C 180,E1 -20658.354,E2 -20658.354} C_VEL
LIN {X 0,Y 224.287,Z 400.43,A -85,B 0,C 180,E1 -20659.591,E2 -20659.591} C_VEL
LIN {X 0,Y 221.724,Z 395.651,A -85,B 0,C 180,E1 -20660.73,E2 -20660.73} C_VEL
LIN {X 0,Y 219.518,Z 392.082,A -85,B 0,C 180,E1 -20661.675,E2 -20661.675} C_VEL
LIN {X 0,Y 218.663,Z 390.366,A -85,B 0,C 180,E1 -20662.061,E2 -20662.061} C_VEL
LIN {X 0,Y 216.419,Z 387.448,A -85,B 0,C 180,E1 -20663.002,E2 -20663.002} C_VEL
LIN {X 0,Y 215.387,Z 384.479,A -85,B 0,C 180,E1 -20663.598,E2 -20663.598} C_VEL
LIN {X 0,Y 214.893,Z 381.352,A -85,B 0,C 180,E1 -20668.448,E2 -20668.448} C_VEL
LIN {X 0,Y 214.579,Z 378.867,A -85,B 0,C 180,E1 -20672.708,E2 -20672.708} C_VEL
LIN {X 0,Y 214.197,Z 376.75,A -85,B 0,C 180,E1 -20676.813,E2 -20676.813} C_VEL
LIN {X 0,Y 213.909,Z 374.895,A -85,B 0,C 180,E1 -20680.819,E2 -20680.819} C_VEL
LIN {X 0,Y 213.947,Z 374.463,A -85,B 0,C 180,E1 -20682.804,E2 -20682.804} C_VEL
LIN {X 0,Y 213.984,Z 374.461,A -85,B 0,C 180,E1 -20686.709,E2 -20686.709} C_VEL
LIN {X 0,Y 214.2,Z 374.434,A -85,B 0,C 180,E1 -20690.558,E2 -20690.558} C_VEL
LIN {X 0,Y 214.252,Z 374.426,A -85,B 0,C 180,E1 -20692.461,E2 -20692.461} C_VEL
LIN {X 0,Y 214.45,Z 374.398,A -85,B 0,C 180,E1 -20698.122,E2 -20698.122} C_VEL
LIN {X 0,Y 214.554,Z 374.379,A -85,B 0,C 180,E1 -20700,E2 -20700} C_VEL
LIN {X 0,Y 214.45,Z 374.397,A -85,B 0,C 180,E1 -20701.878,E2 -20701.878} C_VEL
LIN {X 0,Y 214.252,Z 374.416,A -85,B 0,C 180,E1 -20707.54,E2 -20707.54} C_VEL
LIN {X 0,Y 214.03,Z 374.418,A -85,B 0,C 180,E1 -20711.363,E2 -20711.363} C_VEL
LIN {X 0,Y 213.937,Z 374.445,A -85,B 0,C 180,E1 -20715.237,E2 -20715.237} C_VEL
LIN {X 0,Y 213.839,Z 374.443,A -85,B 0,C 180,E1 -20719.188,E2 -20719.188} C_VEL
LIN {X 0,Y 213.815,Z 374.471,A -85,B 0,C 180,E1 -20723.231,E2 -20723.231} C_VEL
LIN {X 0,Y 213.833,Z 374.444,A -85,B 0,C 180,E1 -20727.45,E2 -20727.45} C_VEL
LIN {X 0,Y 213.773,Z 374.469,A -85,B 0,C 180,E1 -20731.737,E2 -20731.737} C_VEL
LIN {X 0,Y 213.771,Z 374.522,A -85,B 0,C 180,E1 -20736.066,E2 -20736.066} C_VEL
LIN {X 0,Y 214.58,Z 377.033,A -85,B 0,C 180,E1 -20736.532,E2 -20736.532} C_VEL
LIN {X 0,Y 216.767,Z 379.423,A -85,B 0,C 180,E1 -20737.471,E2 -20737.471} C_VEL
LIN {X 0,Y 217.576,Z 380.239,A -85,B 0,C 180,E1 -20737.804,E2 -20737.804} C_VEL
LIN {X 0,Y 219.377,Z 383.301,A -85,B 0,C 180,E1 -20738.661,E2 -20738.661} C_VEL
LIN {X 0,Y 221.005,Z 385.204,A -85,B 0,C 180,E1 -20739.347,E2 -20739.347} C_VEL
LIN {X 0,Y 223.493,Z 388.843,A -85,B 0,C 180,E1 -20740.435,E2 -20740.435} C_VEL
LIN {X 0,Y 229.002,Z 397.915,A -85,B 0,C 180,E1 -20742.934,E2 -20742.934} C_VEL
LIN {X 0,Y 233.264,Z 406.822,A -85,B 0,C 180,E1 -20745.075,E2 -20745.075} C_VEL
LIN {X 0,Y 237.532,Z 418.866,A -85,B 0,C 180,E1 -20747.705,E2 -20747.705} C_VEL
LIN {X 0,Y 240.436,Z 430.307,A -85,B 0,C 180,E1 -20750.11,E2 -20750.11} C_VEL
LIN {X 0,Y 242.201,Z 441.349,A -85,B 0,C 180,E1 -20752.456,E2 -20752.456} C_VEL
LIN {X 0,Y 242.298,Z 442.229,A -85,B 0,C 180,E1 -20752.64,E2 -20752.64} C_VEL
LIN {X 0,Y 238.417,Z 455.129,A -85,B 0,C 180,E1 -20754.654,E2 -20754.654} C_VEL
LIN {X 0,Y 234.339,Z 466.509,A -85,B 0,C 180,E1 -20756.815,E2 -20756.815} C_VEL
LIN {X 0,Y 231.066,Z 475.333,A -85,B 0,C 180,E1 -20758.864,E2 -20758.864} C_VEL
LIN {X 0,Y 226.806,Z 485.792,A -85,B 0,C 180,E1 -20761.799,E2 -20761.799} C_VEL
LIN {X 0,Y 223.044,Z 494.479,A -85,B 0,C 180,E1 -20764.825,E2 -20764.825} C_VEL
LIN {X 0,Y 219.733,Z 501.948,A -85,B 0,C 180,E1 -20768.056,E2 -20768.056} C_VEL
LIN {X 0,Y 216.663,Z 509.102,A -85,B 0,C 180,E1 -20772.051,E2 -20772.051} C_VEL
LIN {X 0,Y 214.524,Z 514.176,A -85,B 0,C 180,E1 -20775.776,E2 -20775.776} C_VEL
LIN {X 0,Y 213.378,Z 517.093,A -85,B 0,C 180,E1 -20778.601,E2 -20778.601} C_VEL
LIN {X 0,Y 212.385,Z 519.941,A -85,B 0,C 180,E1 -20782.393,E2 -20782.393} C_VEL
LIN {X 0,Y 211.955,Z 521.645,A -85,B 0,C 180,E1 -20786.197,E2 -20786.197} C_VEL
LIN {X 0,Y 211.782,Z 522.24,A -85,B 0,C 180,E1 -20789.999,E2 -20789.999} C_VEL
LIN {X 0,Y 211.934,Z 521.682,A -85,B 0,C 180,E1 -20793.802,E2 -20793.802} C_VEL
LIN {X 0,Y 212.384,Z 520.025,A -85,B 0,C 180,E1 -20797.605,E2 -20797.605} C_VEL
LIN {X 0,Y 213.361,Z 517.221,A -85,B 0,C 180,E1 -20801.398,E2 -20801.398} C_VEL
LIN {X 0,Y 214.932,Z 513.2,A -85,B 0,C 180,E1 -20805.164,E2 -20805.164} C_VEL
LIN {X 0,Y 217.256,Z 507.854,A -85,B 0,C 180,E1 -20808.873,E2 -20808.873} C_VEL
LIN {X 0,Y 220.141,Z 501.04,A -85,B 0,C 180,E1 -20812.525,E2 -20812.525} C_VEL
LIN {X 0,Y 223.968,Z 492.508,A -85,B 0,C 180,E1 -20816.059,E2 -20816.059} C_VEL
LIN {X 0,Y 227.809,Z 483.432,A -85,B 0,C 180,E1 -20819.07,E2 -20819.07} C_VEL
LIN {X 0,Y 231.759,Z 473.634,A -85,B 0,C 180,E1 -20821.707,E2 -20821.707} C_VEL
LIN {X 0,Y 235.982,Z 462.191,A -85,B 0,C 180,E1 -20824.203,E2 -20824.203} C_VEL
LIN {X 0,Y 240.149,Z 449.932,A -85,B 0,C 180,E1 -20826.342,E2 -20826.342} C_VEL
LIN {X 0,Y 242.338,Z 442.118,A -85,B 0,C 180,E1 -20827.518,E2 -20827.518} C_VEL
LIN {X 0,Y 240.792,Z 431.779,A -85,B 0,C 180,E1 -20829.708,E2 -20829.708} C_VEL
LIN {X 0,Y 238.019,Z 420.346,A -85,B 0,C 180,E1 -20832.121,E2 -20832.121} C_VEL
LIN {X 0,Y 234.255,Z 409.152,A -85,B 0,C 180,E1 -20834.558,E2 -20834.558} C_VEL
LIN {X 0,Y 230.078,Z 399.793,A -85,B 0,C 180,E1 -20836.734,E2 -20836.734} C_VEL
LIN {X 0,Y 225.72,Z 392.456,A -85,B 0,C 180,E1 -20838.723,E2 -20838.723} C_VEL
LIN {X 0,Y 223.07,Z 388.387,A -85,B 0,C 180,E1 -20839.916,E2 -20839.916} C_VEL
LIN {X 0,Y 220.253,Z 384.242,A -85,B 0,C 180,E1 -20841.155,E2 -20841.155} C_VEL
LIN {X 0,Y 218.108,Z 381.379,A -85,B 0,C 180,E1 -20842.112,E2 -20842.112} C_VEL
LIN {X 0,Y 217.098,Z 379.636,A -85,B 0,C 180,E1 -20842.587,E2 -20842.587} C_VEL
LIN {X 0,Y 214.874,Z 377.502,A -85,B 0,C 180,E1 -20843.522,E2 -20843.522} C_VEL
LIN {X 0,Y 213.857,Z 375.085,A -85,B 0,C 180,E1 -20844.059,E2 -20844.059} C_VEL
LIN {X 0,Y 213.758,Z 374.485,A -85,B 0,C 180,E1 -20844.203,E2 -20844.203} C_VEL
LIN {X 0,Y 213.794,Z 374.469,A -85,B 0,C 180,E1 -20848.724,E2 -20848.724} C_VEL
LIN {X 0,Y 213.824,Z 374.447,A -85,B 0,C 180,E1 -20852.603,E2 -20852.603} C_VEL
LIN {X 0,Y 213.85,Z 374.466,A -85,B 0,C 180,E1 -20856.952,E2 -20856.952} C_VEL
LIN {X 0,Y 213.942,Z 374.46,A -85,B 0,C 180,E1 -20862.803,E2 -20862.803} C_VEL
LIN {X 0,Y 213.953,Z 374.423,A -85,B 0,C 180,E1 -20866.706,E2 -20866.706} C_VEL
LIN {X 0,Y 214.195,Z 374.43,A -85,B 0,C 180,E1 -20870.557,E2 -20870.557} C_VEL
LIN {X 0,Y 214.246,Z 374.422,A -85,B 0,C 180,E1 -20872.46,E2 -20872.46} C_VEL
LIN {X 0,Y 214.445,Z 374.398,A -85,B 0,C 180,E1 -20878.122,E2 -20878.122} C_VEL
LIN {X 0,Y 214.553,Z 374.386,A -85,B 0,C 180,E1 -20880,E2 -20880} C_VEL
LIN {X 0,Y 214.445,Z 374.4,A -85,B 0,C 180,E1 -20881.878,E2 -20881.878} C_VEL
LIN {X 0,Y 214.246,Z 374.424,A -85,B 0,C 180,E1 -20887.54,E2 -20887.54} C_VEL
LIN {X 0,Y 214.04,Z 374.446,A -85,B 0,C 180,E1 -20891.362,E2 -20891.362} C_VEL
LIN {X 0,Y 213.96,Z 374.457,A -85,B 0,C 180,E1 -20897.195,E2 -20897.195} C_VEL
LIN {X 0,Y 214.041,Z 375.852,A -85,B 0,C 180,E1 -20901.173,E2 -20901.173} C_VEL
LIN {X 0,Y 214.354,Z 377.829,A -85,B 0,C 180,E1 -20905.228,E2 -20905.228} C_VEL
LIN {X 0,Y 214.721,Z 380.125,A -85,B 0,C 180,E1 -20909.404,E2 -20909.404} C_VEL
LIN {X 0,Y 215.085,Z 382.769,A -85,B 0,C 180,E1 -20913.744,E2 -20913.744} C_VEL
LIN {X 0,Y 215.368,Z 384.487,A -85,B 0,C 180,E1 -20916.333,E2 -20916.333} C_VEL
LIN {X 0,Y 216.567,Z 387.712,A -85,B 0,C 180,E1 -20916.968,E2 -20916.968} C_VEL
LIN {X 0,Y 219.141,Z 391.092,A -85,B 0,C 180,E1 -20918.049,E2 -20918.049} C_VEL
LIN {X 0,Y 220.925,Z 394.573,A -85,B 0,C 180,E1 -20918.849,E2 -20918.849} C_VEL
LIN {X 0,Y 222.418,Z 396.803,A -85,B 0,C 180,E1 -20919.488,E2 -20919.488} C_VEL
LIN {X 0,Y 224.892,Z 401.324,A -85,B 0,C 180,E1 -20920.572,E2 -20920.572} C_VEL
LIN {X 0,Y 229.454,Z 410.799,A -85,B 0,C 180,E1 -20922.685,E2 -20922.685} C_VEL
LIN {X 0,Y 232.075,Z 418.468,A -85,B 0,C 180,E1 -20924.148,E2 -20924.148} C_VEL
LIN {X 0,Y 234.909,Z 429.909,A -85,B 0,C 180,E1 -20926.201,E2 -20926.201} C_VEL
LIN {X 0,Y 236.753,Z 440.92,A -85,B 0,C 180,E1 -20928.122,E2 -20928.122} C_VEL
LIN {X 0,Y 237.688,Z 451.491,A -85,B 0,C 180,E1 -20930.012,E2 -20930.012} C_VEL
LIN {X 0,Y 237.952,Z 462.872,A -85,B 0,C 180,E1 -20932.127,E2 -20932.127} C_VEL
LIN {X 0,Y 237.686,Z 469.566,A -85,B 0,C 180,E1 -20933.44,E2 -20933.44} C_VEL
LIN {X 0,Y 234.584,Z 478.43,A -85,B 0,C 180,E1 -20934.94,E2 -20934.94} C_VEL
LIN {X 0,Y 232.307,Z 482.961,A -85,B 0,C 180,E1 -20935.7,E2 -20935.7} C_VEL
LIN {X 0,Y 227.077,Z 490.03,A -85,B 0,C 180,E1 -20936.84,E2 -20936.84} C_VEL
LIN {X 0,Y 221.877,Z 496.757,A -85,B 0,C 180,E1 -20938.138,E2 -20938.138} C_VEL
LIN {X 0,Y 219.686,Z 500.609,A -85,B 0,C 180,E1 -20939.137,E2 -20939.137} C_VEL
LIN {X 0,Y 215.557,Z 510.387,A -85,B 0,C 180,E1 -20942.316,E2 -20942.316} C_VEL
LIN {X 0,Y 212.089,Z 518.364,A -85,B 0,C 180,E1 -20945.531,E2 -20945.531} C_VEL
LIN {X 0,Y 208.976,Z 525.83,A -85,B 0,C 180,E1 -20949.322,E2 -20949.322} C_VEL
LIN {X 0,Y 206.732,Z 531.771,A -85,B 0,C 180,E1 -20953.205,E2 -20953.205} C_VEL
LIN {X 0,Y 205.571,Z 535.315,A -85,B 0,C 180,E1 -20956.155,E2 -20956.155} C_VEL
LIN {X 0,Y 204.672,Z 538.907,A -85,B 0,C 180,E1 -20960.115,E2 -20960.115} C_VEL
LIN {X 0,Y 204.473,Z 541.288,A -85,B 0,C 180,E1 -20964.082,E2 -20964.082} C_VEL
LIN {X 0,Y 204.554,Z 542.49,A -85,B 0,C 180,E1 -20968.032,E2 -20968.032} C_VEL
LIN {X 0,Y 204.674,Z 542.653,A -85,B 0,C 180,E1 -20970.001,E2 -20970.001} C_VEL
LIN {X 0,Y 204.472,Z 542.02,A -85,B 0,C 180,E1 -20973.943,E2 -20973.943} C_VEL
LIN {X 0,Y 204.528,Z 540.214,A -85,B 0,C 180,E1 -20977.901,E2 -20977.901} C_VEL
LIN {X 0,Y 205.008,Z 537.219,A -85,B 0,C 180,E1 -20981.871,E2 -20981.871} C_VEL
LIN {X 0,Y 206.276,Z 532.982,A -85,B 0,C 180,E1 -20985.818,E2 -20985.818} C_VEL
LIN {X 0,Y 208.348,Z 527.392,A -85,B 0,C 180,E1 -20989.714,E2 -20989.714} C_VEL
LIN {X 0,Y 211.203,Z 520.299,A -85,B 0,C 180,E1 -20993.536,E2 -20993.536} C_VEL
LIN {X 0,Y 214.577,Z 512.741,A -85,B 0,C 180,E1 -20996.767,E2 -20996.767} C_VEL
LIN {X 0,Y 218.261,Z 503.904,A -85,B 0,C 180,E1 -20999.835,E2 -20999.835} C_VEL
LIN {X 0,Y 222.278,Z 494.353,A -85,B 0,C 180,E1 -21002.515,E2 -21002.515} C_VEL
LIN {X 0,Y 226.608,Z 483.434,A -85,B 0,C 180,E1 -21005.014,E2 -21005.014} C_VEL
LIN {X 0,Y 231.114,Z 471.537,A -85,B 0,C 180,E1 -21007.185,E2 -21007.185} C_VEL
LIN {X 0,Y 231.753,Z 463.929,A -85,B 0,C 180,E1 -21008.716,E2 -21008.716} C_VEL
LIN {X 0,Y 231.615,Z 452.781,A -85,B 0,C 180,E1 -21010.901,E2 -21010.901} C_VEL
LIN {X 0,Y 230.751,Z 441.329,A -85,B 0,C 180,E1 -21013.033,E2 -21013.033} C_VEL
LIN {X 0,Y 228.635,Z 429.034,A -85,B 0,C 180,E1 -21015.32,E2 -21015.32} C_VEL
LIN {X 0,Y 225.883,Z 418.271,A -85,B 0,C 180,E1 -21017.392,E2 -21017.392} C_VEL
LIN {X 0,Y 222.697,Z 410.343,A -85,B 0,C 180,E1 -21019.152,E2 -21019.152} C_VEL
LIN {X 0,Y 219.749,Z 404.591,A -85,B 0,C 180,E1 -21020.593,E2 -21020.593} C_VEL
LIN {X 0,Y 217.879,Z 400.798,A -85,B 0,C 180,E1 -21021.542,E2 -21021.542} C_VEL
LIN {X 0,Y 215.618,Z 396.79,A -85,B 0,C 180,E1 -21022.622,E2 -21022.622} C_VEL
LIN {X 0,Y 212.531,Z 391.79,A -85,B 0,C 180,E1 -21024.105,E2 -21024.105} C_VEL
LIN {X 0,Y 211.599,Z 389.984,A -85,B 0,C 180,E1 -21024.571,E2 -21024.571} C_VEL
LIN {X 0,Y 209.219,Z 387.06,A -85,B 0,C 180,E1 -21025.688,E2 -21025.688} C_VEL
LIN {X 0,Y 208.087,Z 383.883,A -85,B 0,C 180,E1 -21026.423,E2 -21026.423} C_VEL
LIN {X 0,Y 207.65,Z 380.8,A -85,B 0,C 180,E1 -21031.717,E2 -21031.717} C_VEL
LIN {X 0,Y 207.263,Z 378.439,A -85,B 0,C 180,E1 -21036.283,E2 -21036.283} C_VEL
LIN {X 0,Y 206.95,Z 375.807,A -85,B 0,C 180,E1 -21042.204,E2 -21042.204} C_VEL
LIN {X 0,Y 206.871,Z 375.345,A -85,B 0,C 180,E1 -21044.23,E2 -21044.23} C_VEL
LIN {X 0,Y 207.121,Z 375.315,A -85,B 0,C 180,E1 -21049.748,E2 -21049.748} C_VEL
LIN {X 0,Y 207.193,Z 375.307,A -85,B 0,C 180,E1 -21052.202,E2 -21052.202} C_VEL
LIN {X 0,Y 207.387,Z 375.278,A -85,B 0,C 180,E1 -21058.058,E2 -21058.058} C_VEL
LIN {X 0,Y 207.519,Z 375.255,A -85,B 0,C 180,E1 -21060,E2 -21060} C_VEL
LIN {X 0,Y 207.387,Z 375.277,A -85,B 0,C 180,E1 -21061.942,E2 -21061.942} C_VEL
LIN {X 0,Y 207.193,Z 375.297,A -85,B 0,C 180,E1 -21067.798,E2 -21067.798} C_VEL
LIN {X 0,Y 206.949,Z 375.295,A -85,B 0,C 180,E1 -21071.757,E2 -21071.757} C_VEL
LIN {X 0,Y 206.871,Z 375.334,A -85,B 0,C 180,E1 -21075.771,E2 -21075.771} C_VEL
LIN {X 0,Y 206.766,Z 375.318,A -85,B 0,C 180,E1 -21079.871,E2 -21079.871} C_VEL
LIN {X 0,Y 206.751,Z 375.356,A -85,B 0,C 180,E1 -21084.074,E2 -21084.074} C_VEL
LIN {X 0,Y 206.74,Z 375.332,A -85,B 0,C 180,E1 -21088.42,E2 -21088.42} C_VEL
LIN {X 0,Y 206.722,Z 375.525,A -85,B 0,C 180,E1 -21093.317,E2 -21093.317} C_VEL
LIN {X 0,Y 207.621,Z 378.016,A -85,B 0,C 180,E1 -21093.881,E2 -21093.881} C_VEL
LIN {X 0,Y 209.754,Z 380.318,A -85,B 0,C 180,E1 -21094.915,E2 -21094.915} C_VEL
LIN {X 0,Y 210.652,Z 381.052,A -85,B 0,C 180,E1 -21095.322,E2 -21095.322} C_VEL
LIN {X 0,Y 212.388,Z 384.156,A -85,B 0,C 180,E1 -21096.263,E2 -21096.263} C_VEL
LIN {X 0,Y 214.278,Z 386.235,A -85,B 0,C 180,E1 -21097.14,E2 -21097.14} C_VEL
LIN {X 0,Y 216.553,Z 389.706,A -85,B 0,C 180,E1 -21098.261,E2 -21098.261} C_VEL
LIN {X 0,Y 217.962,Z 391.852,A -85,B 0,C 180,E1 -21098.959,E2 -21098.959} C_VEL
LIN {X 0,Y 220.674,Z 396.05,A -85,B 0,C 180,E1 -21100.264,E2 -21100.264} C_VEL
LIN {X 0,Y 224.096,Z 401.721,A -85,B 0,C 180,E1 -21101.955,E2 -21101.955} C_VEL
LIN {X 0,Y 228.488,Z 411.308,A -85,B 0,C 180,E1 -21104.408,E2 -21104.408} C_VEL
LIN {X 0,Y 232.24,Z 422.687,A -85,B 0,C 180,E1 -21107.036,E2 -21107.036} C_VEL
LIN {X 0,Y 234.725,Z 433.467,A -85,B 0,C 180,E1 -21109.444,E2 -21109.444} C_VEL
LIN {X 0,Y 236.237,Z 443.91,A -85,B 0,C 180,E1 -21111.765,E2 -21111.765} C_VEL
LIN {X 0,Y 232.284,Z 456.636,A -85,B 0,C 180,E1 -21113.843,E2 -21113.843} C_VEL
LIN {X 0,Y 227.674,Z 468.774,A -85,B 0,C 180,E1 -21116.245,E2 -21116.245} C_VEL
LIN {X 0,Y 223.679,Z 478.908,A -85,B 0,C 180,E1 -21118.772,E2 -21118.772} C_VEL
LIN {X 0,Y 219.364,Z 488.821,A -85,B 0,C 180,E1 -21121.798,E2 -21121.798} C_VEL
LIN {X 0,Y 215.574,Z 497.035,A -85,B 0,C 180,E1 -21124.923,E2 -21124.923} C_VEL
LIN {X 0,Y 211.99,Z 504.738,A -85,B 0,C 180,E1 -21128.611,E2 -21128.611} C_VEL
LIN {X 0,Y 209.199,Z 510.857,A -85,B 0,C 180,E1 -21132.4,E2 -21132.4} C_VEL
LIN {X 0,Y 207.197,Z 515.568,A -85,B 0,C 180,E1 -21136.264,E2 -21136.264} C_VEL
LIN {X 0,Y 205.793,Z 519.013,A -85,B 0,C 180,E1 -21140.167,E2 -21140.167} C_VEL
LIN {X 0,Y 205.035,Z 521.281,A -85,B 0,C 180,E1 -21144.097,E2 -21144.097} C_VEL
LIN {X 0,Y 204.77,Z 522.432,A -85,B 0,C 180,E1 -21148.032,E2 -21148.032} C_VEL
LIN {X 0,Y 204.768,Z 522.443,A -85,B 0,C 180,E1 -21151.966,E2 -21151.966} C_VEL
LIN {X 0,Y 205.145,Z 521.091,A -85,B 0,C 180,E1 -21156.533,E2 -21156.533} C_VEL
LIN {X 0,Y 205.787,Z 519.119,A -85,B 0,C 180,E1 -21159.831,E2 -21159.831} C_VEL
LIN {X 0,Y 207.155,Z 515.716,A -85,B 0,C 180,E1 -21163.737,E2 -21163.737} C_VEL
LIN {X 0,Y 209.151,Z 511.051,A -85,B 0,C 180,E1 -21167.602,E2 -21167.602} C_VEL
LIN {X 0,Y 211.908,Z 504.994,A -85,B 0,C 180,E1 -21171.396,E2 -21171.396} C_VEL
LIN {X 0,Y 215.503,Z 497.351,A -85,B 0,C 180,E1 -21175.084,E2 -21175.084} C_VEL
LIN {X 0,Y 219.287,Z 489.191,A -85,B 0,C 180,E1 -21178.211,E2 -21178.211} C_VEL
LIN {X 0,Y 223.584,Z 479.352,A -85,B 0,C 180,E1 -21181.241,E2 -21181.241} C_VEL
LIN {X 0,Y 227.57,Z 469.265,A -85,B 0,C 180,E1 -21183.771,E2 -21183.771} C_VEL
LIN {X 0,Y 231.748,Z 458.288,A -85,B 0,C 180,E1 -21185.984,E2 -21185.984} C_VEL
LIN {X 0,Y 235.585,Z 446.718,A -85,B 0,C 180,E1 -21187.912,E2 -21187.912} C_VEL
LIN {X 0,Y 236.31,Z 444.256,A -85,B 0,C 180,E1 -21188.295,E2 -21188.295} C_VEL
LIN {X 0,Y 234.87,Z 433.901,A -85,B 0,C 180,E1 -21190.599,E2 -21190.599} C_VEL
LIN {X 0,Y 232.286,Z 422.74,A -85,B 0,C 180,E1 -21193.104,E2 -21193.104} C_VEL
LIN {X 0,Y 229.384,Z 413.594,A -85,B 0,C 180,E1 -21195.195,E2 -21195.195} C_VEL
LIN {X 0,Y 225.926,Z 405.327,A -85,B 0,C 180,E1 -21197.238,E2 -21197.238} C_VEL
LIN {X 0,Y 221.703,Z 397.713,A -85,B 0,C 180,E1 -21199.396,E2 -21199.396} C_VEL
LIN {X 0,Y 218.969,Z 393.364,A -85,B 0,C 180,E1 -21200.736,E2 -21200.736} C_VEL
LIN {X 0,Y 216.545,Z 389.698,A -85,B 0,C 180,E1 -21201.928,E2 -21201.928} C_VEL
LIN {X 0,Y 214.133,Z 385.932,A -85,B 0,C 180,E1 -21203.13,E2 -21203.13} C_VEL
LIN {X 0,Y 211.483,Z 382.835,A -85,B 0,C 180,E1 -21204.397,E2 -21204.397} C_VEL
LIN {X 0,Y 210.379,Z 380.715,A -85,B 0,C 180,E1 -21205.011,E2 -21205.011} C_VEL
LIN {X 0,Y 207.91,Z 378.489,A -85,B 0,C 180,E1 -21206.172,E2 -21206.172} C_VEL
LIN {X 0,Y 206.863,Z 376.234,A -85,B 0,C 180,E1 -21206.781,E2 -21206.781} C_VEL
LIN {X 0,Y 206.695,Z 375.34,A -85,B 0,C 180,E1 -21206.969,E2 -21206.969} C_VEL
LIN {X 0,Y 206.743,Z 375.336,A -85,B 0,C 180,E1 -21211.581,E2 -21211.581} C_VEL
LIN {X 0,Y 206.784,Z 375.35,A -85,B 0,C 180,E1 -21216.583,E2 -21216.583} C_VEL
LIN {X 0,Y 206.872,Z 375.334,A -85,B 0,C 180,E1 -21222.196,E2 -21222.196} C_VEL
LIN {X 0,Y 206.895,Z 375.303,A -85,B 0,C 180,E1 -21226.244,E2 -21226.244} C_VEL
LIN {X 0,Y 207.131,Z 375.308,A -85,B 0,C 180,E1 -21230.232,E2 -21230.232} C_VEL
LIN {X 0,Y 207.187,Z 375.3,A -85,B 0,C 180,E1 -21232.202,E2 -21232.202} C_VEL
LIN {X 0,Y 207.382,Z 375.278,A -85,B 0,C 180,E1 -21238.058,E2 -21238.058} C_VEL
LIN {X 0,Y 207.517,Z 375.262,A -85,B 0,C 180,E1 -21240,E2 -21240} C_VEL
LIN {X 0,Y 207.087,Z 375.317,A -85,B 0,C 180,E1 -21243.892,E2 -21243.892} C_VEL
LIN {X 0,Y 207.187,Z 375.302,A -85,B 0,C 180,E1 -21247.798,E2 -21247.798} C_VEL
LIN {X 0,Y 206.973,Z 375.323,A -85,B 0,C 180,E1 -21251.755,E2 -21251.755} C_VEL
LIN {X 0,Y 206.87,Z 375.334,A -85,B 0,C 180,E1 -21255.77,E2 -21255.77} C_VEL
LIN {X 0,Y 206.947,Z 375.961,A -85,B 0,C 180,E1 -21258.034,E2 -21258.034} C_VEL
LIN {X 0,Y 207.296,Z 378.497,A -85,B 0,C 180,E1 -21263.742,E2 -21263.742} C_VEL
LIN {X 0,Y 207.654,Z 380.904,A -85,B 0,C 180,E1 -21268.364,E2 -21268.364} C_VEL
LIN {X 0,Y 208.138,Z 384.095,A -85,B 0,C 180,E1 -21273.567,E2 -21273.567} C_VEL
LIN {X 0,Y 209.174,Z 386.955,A -85,B 0,C 180,E1 -21274.175,E2 -21274.175} C_VEL
LIN {X 0,Y 211.593,Z 389.973,A -85,B 0,C 180,E1 -21275.32,E2 -21275.32} C_VEL
LIN {X 0,Y 212.324,Z 391.264,A -85,B 0,C 180,E1 -21275.68,E2 -21275.68} C_VEL
LIN {X 0,Y 214.348,Z 394.88,A -85,B 0,C 180,E1 -21276.68,E2 -21276.68} C_VEL
LIN {X 0,Y 215.553,Z 396.6,A -85,B 0,C 180,E1 -21277.244,E2 -21277.244} C_VEL
LIN {X 0,Y 217.902,Z 400.855,A -85,B 0,C 180,E1 -21278.379,E2 -21278.379} C_VEL
LIN {X 0,Y 221.538,Z 408,A -85,B 0,C 180,E1 -21280.195,E2 -21280.195} C_VEL
LIN {X 0,Y 225.033,Z 415.815,A -85,B 0,C 180,E1 -21282.029,E2 -21282.029} C_VEL
LIN {X 0,Y 227.448,Z 423.59,A -85,B 0,C 180,E1 -21283.598,E2 -21283.598} C_VEL
LIN {X 0,Y 230.228,Z 437.163,A -85,B 0,C 180,E1 -21286.151,E2 -21286.151} C_VEL
LIN {X 0,Y 231.655,Z 450.643,A -85,B 0,C 180,E1 -21288.666,E2 -21288.666} C_VEL
LIN {X 0,Y 231.804,Z 464.184,A -85,B 0,C 180,E1 -21291.292,E2 -21291.292} C_VEL
LIN {X 0,Y 231.473,Z 470.593,A -85,B 0,C 180,E1 -21292.611,E2 -21292.611} C_VEL
LIN {X 0,Y 227.342,Z 481.667,A -85,B 0,C 180,E1 -21294.576,E2 -21294.576} C_VEL
LIN {X 0,Y 222.923,Z 492.878,A -85,B 0,C 180,E1 -21297.056,E2 -21297.056} C_VEL
LIN {X 0,Y 219.686,Z 500.609,A -85,B 0,C 180,E1 -21299.137,E2 -21299.137} C_VEL
LIN {X 0,Y 217.526,Z 504.38,A -85,B 0,C 180,E1 -21300.196,E2 -21300.196} C_VEL
LIN {X 0,Y 212.439,Z 510.172,A -85,B 0,C 180,E1 -21301.856,E2 -21301.856} C_VEL
LIN {X 0,Y 207.381,Z 515.554,A -85,B 0,C 180,E1 -21303.673,E2 -21303.673} C_VEL
LIN {X 0,Y 205.315,Z 518.568,A -85,B 0,C 180,E1 -21304.962,E2 -21304.962} C_VEL
LIN {X 0,Y 202.269,Z 525.479,A -85,B 0,C 180,E1 -21308.604,E2 -21308.604} C_VEL
LIN {X 0,Y 199.874,Z 531.42,A -85,B 0,C 180,E1 -21312.611,E2 -21312.611} C_VEL
LIN {X 0,Y 198.601,Z 534.963,A -85,B 0,C 180,E1 -21315.659,E2 -21315.659} C_VEL
LIN {X 0,Y 197.628,Z 538.557,A -85,B 0,C 180,E1 -21319.759,E2 -21319.759} C_VEL
LIN {X 0,Y 197.372,Z 540.938,A -85,B 0,C 180,E1 -21323.869,E2 -21323.869} C_VEL
LIN {X 0,Y 197.468,Z 542.143,A -85,B 0,C 180,E1 -21327.961,E2 -21327.961} C_VEL
LIN {X 0,Y 197.586,Z 542.306,A -85,B 0,C 180,E1 -21330.001,E2 -21330.001} C_VEL
LIN {X 0,Y 197.393,Z 541.672,A -85,B 0,C 180,E1 -21334.084,E2 -21334.084} C_VEL
LIN {X 0,Y 197.45,Z 539.864,A -85,B 0,C 180,E1 -21338.186,E2 -21338.186} C_VEL
LIN {X 0,Y 197.993,Z 536.867,A -85,B 0,C 180,E1 -21342.298,E2 -21342.298} C_VEL
LIN {X 0,Y 199.377,Z 532.629,A -85,B 0,C 180,E1 -21346.38,E2 -21346.38} C_VEL
LIN {X 0,Y 201.58,Z 527.037,A -85,B 0,C 180,E1 -21350.405,E2 -21350.405} C_VEL
LIN {X 0,Y 204.62,Z 519.945,A -85,B 0,C 180,E1 -21354.341,E2 -21354.341} C_VEL
LIN {X 0,Y 208.166,Z 512.386,A -85,B 0,C 180,E1 -21357.661,E2 -21357.661} C_VEL
LIN {X 0,Y 212.178,Z 503.276,A -85,B 0,C 180,E1 -21360.892,E2 -21360.892} C_VEL
LIN {X 0,Y 216.978,Z 492.35,A -85,B 0,C 180,E1 -21363.969,E2 -21363.969} C_VEL
LIN {X 0,Y 221.578,Z 481.115,A -85,B 0,C 180,E1 -21366.493,E2 -21366.493} C_VEL
LIN {X 0,Y 224.982,Z 472.462,A -85,B 0,C 180,E1 -21368.071,E2 -21368.071} C_VEL
LIN {X 0,Y 225.778,Z 462.217,A -85,B 0,C 180,E1 -21370.234,E2 -21370.234} C_VEL
LIN {X 0,Y 225.448,Z 449.021,A -85,B 0,C 180,E1 -21372.899,E2 -21372.899} C_VEL
LIN {X 0,Y 224.326,Z 438.183,A -85,B 0,C 180,E1 -21375.02,E2 -21375.02} C_VEL
LIN {X 0,Y 222.274,Z 427.41,A -85,B 0,C 180,E1 -21377.171,E2 -21377.171} C_VEL
LIN {X 0,Y 220.047,Z 419.332,A -85,B 0,C 180,E1 -21378.874,E2 -21378.874} C_VEL
LIN {X 0,Y 216.352,Z 410.822,A -85,B 0,C 180,E1 -21381.019,E2 -21381.019} C_VEL
LIN {X 0,Y 213.5,Z 405.254,A -85,B 0,C 180,E1 -21382.558,E2 -21382.558} C_VEL
LIN {X 0,Y 211.145,Z 400.745,A -85,B 0,C 180,E1 -21383.859,E2 -21383.859} C_VEL
LIN {X 0,Y 208.817,Z 396.616,A -85,B 0,C 180,E1 -21385.1,E2 -21385.1} C_VEL
LIN {X 0,Y 208.005,Z 395.338,A -85,B 0,C 180,E1 -21385.533,E2 -21385.533} C_VEL
LIN {X 0,Y 205.681,Z 391.807,A -85,B 0,C 180,E1 -21386.785,E2 -21386.785} C_VEL
LIN {X 0,Y 204.641,Z 389.619,A -85,B 0,C 180,E1 -21387.389,E2 -21387.389} C_VEL
LIN {X 0,Y 202.147,Z 386.799,A -85,B 0,C 180,E1 -21388.713,E2 -21388.713} C_VEL
LIN {X 0,Y 200.912,Z 383.761,A -85,B 0,C 180,E1 -21389.522,E2 -21389.522} C_VEL
LIN {X 0,Y 200.816,Z 383.278,A -85,B 0,C 180,E1 -21389.651,E2 -21389.651} C_VEL
LIN {X 0,Y 200.562,Z 381.528,A -85,B 0,C 180,E1 -21392.901,E2 -21392.901} C_VEL
LIN {X 0,Y 200.212,Z 379.415,A -85,B 0,C 180,E1 -21397.286,E2 -21397.286} C_VEL
LIN {X 0,Y 199.997,Z 377.55,A -85,B 0,C 180,E1 -21401.587,E2 -21401.587} C_VEL
LIN {X 0,Y 199.852,Z 376.22,A -85,B 0,C 180,E1 -21405.75,E2 -21405.75} C_VEL
LIN {X 0,Y 200.079,Z 376.192,A -85,B 0,C 180,E1 -21409.885,E2 -21409.885} C_VEL
LIN {X 0,Y 200.136,Z 376.185,A -85,B 0,C 180,E1 -21411.926,E2 -21411.926} C_VEL
LIN {X 0,Y 200.326,Z 376.157,A -85,B 0,C 180,E1 -21417.99,E2 -21417.99} C_VEL
LIN {X 0,Y 200.483,Z 376.131,A -85,B 0,C 180,E1 -21420,E2 -21420} C_VEL
LIN {X 0,Y 200.037,Z 376.188,A -85,B 0,C 180,E1 -21424.03,E2 -21424.03} C_VEL
LIN {X 0,Y 200.137,Z 376.178,A -85,B 0,C 180,E1 -21428.075,E2 -21428.075} C_VEL
LIN {X 0,Y 200.072,Z 376.169,A -85,B 0,C 180,E1 -21430.398,E2 -21430.398} C_VEL
LIN {X 0,Y 199.809,Z 376.22,A -85,B 0,C 180,E1 -21436.343,E2 -21436.343} C_VEL
LIN {X 0,Y 199.685,Z 376.199,A -85,B 0,C 180,E1 -21440.607,E2 -21440.607} C_VEL
LIN {X 0,Y 199.668,Z 376.227,A -85,B 0,C 180,E1 -21444.985,E2 -21444.985} C_VEL
LIN {X 0,Y 199.665,Z 376.232,A -85,B 0,C 180,E1 -21449.814,E2 -21449.814} C_VEL
LIN {X 0,Y 199.663,Z 376.34,A -85,B 0,C 180,E1 -21450.106,E2 -21450.106} C_VEL
LIN {X 0,Y 200.55,Z 378.89,A -85,B 0,C 180,E1 -21450.759,E2 -21450.759} C_VEL
LIN {X 0,Y 202.535,Z 381.079,A -85,B 0,C 180,E1 -21451.879,E2 -21451.879} C_VEL
LIN {X 0,Y 203.848,Z 382.057,A -85,B 0,C 180,E1 -21452.56,E2 -21452.56} C_VEL
LIN {X 0,Y 205.592,Z 385.188,A -85,B 0,C 180,E1 -21453.637,E2 -21453.637} C_VEL
LIN {X 0,Y 207.573,Z 387.292,A -85,B 0,C 180,E1 -21454.668,E2 -21454.668} C_VEL
LIN {X 0,Y 209.979,Z 390.935,A -85,B 0,C 180,E1 -21456.003,E2 -21456.003} C_VEL
LIN {X 0,Y 211.185,Z 392.643,A -85,B 0,C 180,E1 -21456.651,E2 -21456.651} C_VEL
LIN {X 0,Y 214.488,Z 397.729,A -85,B 0,C 180,E1 -21458.421,E2 -21458.421} C_VEL
LIN {X 0,Y 219.315,Z 406.025,A -85,B 0,C 180,E1 -21461.066,E2 -21461.066} C_VEL
LIN {X 0,Y 223.035,Z 414.161,A -85,B 0,C 180,E1 -21463.327,E2 -21463.327} C_VEL
LIN {X 0,Y 226.406,Z 424.535,A -85,B 0,C 180,E1 -21465.88,E2 -21465.88} C_VEL
LIN {X 0,Y 228.684,Z 434.764,A -85,B 0,C 180,E1 -21468.307,E2 -21468.307} C_VEL
LIN {X 0,Y 230.172,Z 445.538,A -85,B 0,C 180,E1 -21470.842,E2 -21470.842} C_VEL
LIN {X 0,Y 228.828,Z 450.442,A -85,B 0,C 180,E1 -21471.652,E2 -21471.652} C_VEL
LIN {X 0,Y 224.514,Z 462.307,A -85,B 0,C 180,E1 -21473.782,E2 -21473.782} C_VEL
LIN {X 0,Y 220.351,Z 472.508,A -85,B 0,C 180,E1 -21476.023,E2 -21476.023} C_VEL
LIN {X 0,Y 216.255,Z 482.249,A -85,B 0,C 180,E1 -21478.668,E2 -21478.668} C_VEL
LIN {X 0,Y 211.894,Z 491.647,A -85,B 0,C 180,E1 -21481.794,E2 -21481.794} C_VEL
LIN {X 0,Y 208.129,Z 499.461,A -85,B 0,C 180,E1 -21485.032,E2 -21485.032} C_VEL
LIN {X 0,Y 204.627,Z 506.741,A -85,B 0,C 180,E1 -21488.86,E2 -21488.86} C_VEL
LIN {X 0,Y 201.798,Z 512.512,A -85,B 0,C 180,E1 -21492.78,E2 -21492.78} C_VEL
LIN {X 0,Y 200.304,Z 515.917,A -85,B 0,C 180,E1 -21495.781,E2 -21495.781} C_VEL
LIN {X 0,Y 198.787,Z 519.363,A -85,B 0,C 180,E1 -21499.817,E2 -21499.817} C_VEL
LIN {X 0,Y 197.999,Z 521.628,A -85,B 0,C 180,E1 -21503.886,E2 -21503.886} C_VEL
LIN {X 0,Y 197.687,Z 522.779,A -85,B 0,C 180,E1 -21507.962,E2 -21507.962} C_VEL
LIN {X 0,Y 197.684,Z 522.791,A -85,B 0,C 180,E1 -21512.037,E2 -21512.037} C_VEL
LIN {X 0,Y 198.036,Z 521.562,A -85,B 0,C 180,E1 -21516.444,E2 -21516.444} C_VEL
LIN {X 0,Y 198.781,Z 519.467,A -85,B 0,C 180,E1 -21520.181,E2 -21520.181} C_VEL
LIN {X 0,Y 200.247,Z 516.064,A -85,B 0,C 180,E1 -21524.221,E2 -21524.221} C_VEL
LIN {X 0,Y 202.389,Z 511.398,A -85,B 0,C 180,E1 -21528.211,E2 -21528.211} C_VEL
LIN {X 0,Y 205.28,Z 505.343,A -85,B 0,C 180,E1 -21532.122,E2 -21532.122} C_VEL
LIN {X 0,Y 209.099,Z 497.697,A -85,B 0,C 180,E1 -21535.908,E2 -21535.908} C_VEL
LIN {X 0,Y 213.03,Z 489.539,A -85,B 0,C 180,E1 -21539.117,E2 -21539.117} C_VEL
LIN {X 0,Y 217.54,Z 479.698,A -85,B 0,C 180,E1 -21542.212,E2 -21542.212} C_VEL
LIN {X 0,Y 221.701,Z 469.61,A -85,B 0,C 180,E1 -21544.791,E2 -21544.791} C_VEL
LIN {X 0,Y 226.064,Z 458.632,A -85,B 0,C 180,E1 -21547.037,E2 -21547.037} C_VEL
LIN {X 0,Y 230.135,Z 446.745,A -85,B 0,C 180,E1 -21549.046,E2 -21549.046} C_VEL
LIN {X 0,Y 229.63,Z 440.134,A -85,B 0,C 180,E1 -21550.568,E2 -21550.568} C_VEL
LIN {X 0,Y 227.635,Z 429.247,A -85,B 0,C 180,E1 -21553.136,E2 -21553.136} C_VEL
LIN {X 0,Y 224.762,Z 418.921,A -85,B 0,C 180,E1 -21555.634,E2 -21555.634} C_VEL
LIN {X 0,Y 221.801,Z 411.007,A -85,B 0,C 180,E1 -21557.675,E2 -21557.675} C_VEL
LIN {X 0,Y 218.039,Z 403.528,A -85,B 0,C 180,E1 -21559.86,E2 -21559.86} C_VEL
LIN {X 0,Y 212.963,Z 395.319,A -85,B 0,C 180,E1 -21562.595,E2 -21562.595} C_VEL
LIN {X 0,Y 210.262,Z 391.224,A -85,B 0,C 180,E1 -21564.053,E2 -21564.053} C_VEL
LIN {X 0,Y 207.873,Z 387.869,A -85,B 0,C 180,E1 -21565.36,E2 -21565.36} C_VEL
LIN {X 0,Y 207.092,Z 386.618,A -85,B 0,C 180,E1 -21565.8,E2 -21565.8} C_VEL
LIN {X 0,Y 204.848,Z 384.162,A -85,B 0,C 180,E1 -21566.999,E2 -21566.999} C_VEL
LIN {X 0,Y 203.661,Z 381.73,A -85,B 0,C 180,E1 -21567.773,E2 -21567.773} C_VEL
LIN {X 0,Y 201.223,Z 379.847,A -85,B 0,C 180,E1 -21569.064,E2 -21569.064} C_VEL
LIN {X 0,Y 199.968,Z 377.554,A -85,B 0,C 180,E1 -21569.872,E2 -21569.872} C_VEL
LIN {X 0,Y 199.672,Z 376.236,A -85,B 0,C 180,E1 -21570.187,E2 -21570.187} C_VEL
LIN {X 0,Y 199.671,Z 376.225,A -85,B 0,C 180,E1 -21575.015,E2 -21575.015} C_VEL
LIN {X 0,Y 199.698,Z 376.2,A -85,B 0,C 180,E1 -21579.394,E2 -21579.394} C_VEL
LIN {X 0,Y 199.803,Z 376.219,A -85,B 0,C 180,E1 -21583.656,E2 -21583.656} C_VEL
LIN {X 0,Y 200.066,Z 376.178,A -85,B 0,C 180,E1 -21589.602,E2 -21589.602} C_VEL
LIN {X 0,Y 200.131,Z 376.179,A -85,B 0,C 180,E1 -21591.925,E2 -21591.925} C_VEL
LIN {X 0,Y 200.321,Z 376.158,A -85,B 0,C 180,E1 -21597.989,E2 -21597.989} C_VEL
LIN {X 0,Y 200.481,Z 376.139,A -85,B 0,C 180,E1 -21600,E2 -21600} C_VEL
LIN {X 0,Y 200.032,Z 376.195,A -85,B 0,C 180,E1 -21604.029,E2 -21604.029} C_VEL
LIN {X 0,Y 200.13,Z 376.181,A -85,B 0,C 180,E1 -21608.075,E2 -21608.075} C_VEL
LIN {X 0,Y 199.904,Z 376.201,A -85,B 0,C 180,E1 -21612.177,E2 -21612.177} C_VEL
LIN {X 0,Y 199.835,Z 376.217,A -85,B 0,C 180,E1 -21614.252,E2 -21614.252} C_VEL
LIN {X 0,Y 200.017,Z 377.617,A -85,B 0,C 180,E1 -21618.435,E2 -21618.435} C_VEL
LIN {X 0,Y 200.355,Z 380.111,A -85,B 0,C 180,E1 -21624.216,E2 -21624.216} C_VEL
LIN {X 0,Y 200.708,Z 382.534,A -85,B 0,C 180,E1 -21628.91,E2 -21628.91} C_VEL
LIN {X 0,Y 200.831,Z 383.343,A -85,B 0,C 180,E1 -21630.274,E2 -21630.274} C_VEL
LIN {X 0,Y 201.852,Z 386.223,A -85,B 0,C 180,E1 -21630.974,E2 -21630.974} C_VEL
LIN {X 0,Y 204.215,Z 389.248,A -85,B 0,C 180,E1 -21632.275,E2 -21632.275} C_VEL
LIN {X 0,Y 205.045,Z 390.255,A -85,B 0,C 180,E1 -21632.71,E2 -21632.71} C_VEL
LIN {X 0,Y 206.923,Z 393.932,A -85,B 0,C 180,E1 -21633.791,E2 -21633.791} C_VEL
LIN {X 0,Y 208.875,Z 396.641,A -85,B 0,C 180,E1 -21634.816,E2 -21634.816} C_VEL
LIN {X 0,Y 211.079,Z 400.656,A -85,B 0,C 180,E1 -21636.006,E2 -21636.006} C_VEL
LIN {X 0,Y 212.351,Z 403.045,A -85,B 0,C 180,E1 -21636.712,E2 -21636.712} C_VEL
LIN {X 0,Y 215.033,Z 408.168,A -85,B 0,C 180,E1 -21638.164,E2 -21638.164} C_VEL
LIN {X 0,Y 218.924,Z 416.447,A -85,B 0,C 180,E1 -21640.347,E2 -21640.347} C_VEL
LIN {X 0,Y 221.548,Z 424.004,A -85,B 0,C 180,E1 -21642.077,E2 -21642.077} C_VEL
LIN {X 0,Y 223.881,Z 435.052,A -85,B 0,C 180,E1 -21644.304,E2 -21644.304} C_VEL
LIN {X 0,Y 225.198,Z 444.883,A -85,B 0,C 180,E1 -21646.241,E2 -21646.241} C_VEL
LIN {X 0,Y 225.827,Z 456.407,A -85,B 0,C 180,E1 -21648.528,E2 -21648.528} C_VEL
LIN {X 0,Y 225.563,Z 467.789,A -85,B 0,C 180,E1 -21650.883,E2 -21650.883} C_VEL
LIN {X 0,Y 225.016,Z 472.609,A -85,B 0,C 180,E1 -21651.914,E2 -21651.914} C_VEL
LIN {X 0,Y 220.768,Z 483.287,A -85,B 0,C 180,E1 -21653.92,E2 -21653.92} C_VEL
LIN {X 0,Y 216.221,Z 494.171,A -85,B 0,C 180,E1 -21656.458,E2 -21656.458} C_VEL
LIN {X 0,Y 212.064,Z 503.693,A -85,B 0,C 180,E1 -21659.202,E2 -21659.202} C_VEL
LIN {X 0,Y 208.191,Z 512.512,A -85,B 0,C 180,E1 -21662.345,E2 -21662.345} C_VEL
LIN {X 0,Y 205.315,Z 518.568,A -85,B 0,C 180,E1 -21664.962,E2 -21664.962} C_VEL
LIN {X 0,Y 203.334,Z 521.452,A -85,B 0,C 180,E1 -21666.304,E2 -21666.304} C_VEL
LIN {X 0,Y 198.682,Z 525.727,A -85,B 0,C 180,E1 -21668.481,E2 -21668.481} C_VEL
LIN {X 0,Y 194.306,Z 529.538,A -85,B 0,C 180,E1 -21670.827,E2 -21670.827} C_VEL
LIN {X 0,Y 192.798,Z 531.591,A -85,B 0,C 180,E1 -21672.403,E2 -21672.403} C_VEL
LIN {X 0,Y 191.657,Z 534.612,A -85,B 0,C 180,E1 -21675.127,E2 -21675.127} C_VEL
LIN {X 0,Y 190.585,Z 538.206,A -85,B 0,C 180,E1 -21679.376,E2 -21679.376} C_VEL
LIN {X 0,Y 190.284,Z 540.589,A -85,B 0,C 180,E1 -21683.639,E2 -21683.639} C_VEL
LIN {X 0,Y 190.315,Z 541.338,A -85,B 0,C 180,E1 -21685.765,E2 -21685.765} C_VEL
LIN {X 0,Y 190.499,Z 541.958,A -85,B 0,C 180,E1 -21690.001,E2 -21690.001} C_VEL
LIN {X 0,Y 190.329,Z 541.273,A -85,B 0,C 180,E1 -21694.451,E2 -21694.451} C_VEL
LIN {X 0,Y 190.368,Z 539.512,A -85,B 0,C 180,E1 -21698.493,E2 -21698.493} C_VEL
LIN {X 0,Y 190.988,Z 536.515,A -85,B 0,C 180,E1 -21702.756,E2 -21702.756} C_VEL
LIN {X 0,Y 192.507,Z 532.276,A -85,B 0,C 180,E1 -21706.982,E2 -21706.982} C_VEL
LIN {X 0,Y 194.848,Z 526.683,A -85,B 0,C 180,E1 -21711.144,E2 -21711.144} C_VEL
LIN {X 0,Y 198.09,Z 519.591,A -85,B 0,C 180,E1 -21715.199,E2 -21715.199} C_VEL
LIN {X 0,Y 201.809,Z 512.03,A -85,B 0,C 180,E1 -21718.611,E2 -21718.611} C_VEL
LIN {X 0,Y 206.056,Z 502.922,A -85,B 0,C 180,E1 -21721.916,E2 -21721.916} C_VEL
LIN {X 0,Y 211.08,Z 491.997,A -85,B 0,C 180,E1 -21725.055,E2 -21725.055} C_VEL
LIN {X 0,Y 215.903,Z 480.763,A -85,B 0,C 180,E1 -21727.615,E2 -21727.615} C_VEL
LIN {X 0,Y 218.782,Z 473.75,A -85,B 0,C 180,E1 -21728.941,E2 -21728.941} C_VEL
LIN {X 0,Y 219.641,Z 465.8,A -85,B 0,C 180,E1 -21730.69,E2 -21730.69} C_VEL
LIN {X 0,Y 219.805,Z 453.94,A -85,B 0,C 180,E1 -21733.244,E2 -21733.244} C_VEL
LIN {X 0,Y 219.096,Z 443.381,A -85,B 0,C 180,E1 -21735.428,E2 -21735.428} C_VEL
LIN {X 0,Y 217.304,Z 431.635,A -85,B 0,C 180,E1 -21737.911,E2 -21737.911} C_VEL
LIN {X 0,Y 215.762,Z 425.128,A -85,B 0,C 180,E1 -21739.349,E2 -21739.349} C_VEL
LIN {X 0,Y 212.308,Z 416.1,A -85,B 0,C 180,E1 -21741.691,E2 -21741.691} C_VEL
LIN {X 0,Y 209.072,Z 409.423,A -85,B 0,C 180,E1 -21743.658,E2 -21743.658} C_VEL
LIN {X 0,Y 207.19,Z 405.735,A -85,B 0,C 180,E1 -21744.785,E2 -21744.785} C_VEL
LIN {X 0,Y 204.712,Z 400.998,A -85,B 0,C 180,E1 -21746.313,E2 -21746.313} C_VEL
LIN {X 0,Y 202.237,Z 396.915,A -85,B 0,C 180,E1 -21747.777,E2 -21747.777} C_VEL
LIN {X 0,Y 201.432,Z 395.338,A -85,B 0,C 180,E1 -21748.296,E2 -21748.296} C_VEL
LIN {X 0,Y 198.995,Z 391.961,A -85,B 0,C 180,E1 -21749.783,E2 -21749.783} C_VEL
LIN {X 0,Y 197.767,Z 389.258,A -85,B 0,C 180,E1 -21750.62,E2 -21750.62} C_VEL
LIN {X 0,Y 194.991,Z 386.22,A -85,B 0,C 180,E1 -21752.352,E2 -21752.352} C_VEL
LIN {X 0,Y 193.648,Z 383.133,A -85,B 0,C 180,E1 -21753.386,E2 -21753.386} C_VEL
LIN {X 0,Y 193.536,Z 382.572,A -85,B 0,C 180,E1 -21753.587,E2 -21753.587} C_VEL
LIN {X 0,Y 193.141,Z 380.249,A -85,B 0,C 180,E1 -21758.662,E2 -21758.662} C_VEL
LIN {X 0,Y 192.966,Z 378.477,A -85,B 0,C 180,E1 -21763.06,E2 -21763.06} C_VEL
LIN {X 0,Y 192.857,Z 377.092,A -85,B 0,C 180,E1 -21767.371,E2 -21767.371} C_VEL
LIN {X 0,Y 193.083,Z 377.063,A -85,B 0,C 180,E1 -21771.628,E2 -21771.628} C_VEL
LIN {X 0,Y 193.268,Z 377.036,A -85,B 0,C 180,E1 -21777.916,E2 -21777.916} C_VEL
LIN {X 0,Y 193.447,Z 377.007,A -85,B 0,C 180,E1 -21780,E2 -21780} C_VEL
LIN {X 0,Y 192.984,Z 377.067,A -85,B 0,C 180,E1 -21784.177,E2 -21784.177} C_VEL
LIN {X 0,Y 193.083,Z 377.059,A -85,B 0,C 180,E1 -21788.372,E2 -21788.372} C_VEL
LIN {X 0,Y 193.014,Z 377.044,A -85,B 0,C 180,E1 -21790.538,E2 -21790.538} C_VEL
LIN {X 0,Y 192.761,Z 377.098,A -85,B 0,C 180,E1 -21796.959,E2 -21796.959} C_VEL
LIN {X 0,Y 192.619,Z 377.082,A -85,B 0,C 180,E1 -21801.4,E2 -21801.4} C_VEL
LIN {X 0,Y 192.651,Z 377.111,A -85,B 0,C 180,E1 -21804.213,E2 -21804.213} C_VEL
LIN {X 0,Y 192.603,Z 377.128,A -85,B 0,C 180,E1 -21806.26,E2 -21806.26} C_VEL
LIN {X 0,Y 193.363,Z 379.472,A -85,B 0,C 180,E1 -21806.949,E2 -21806.949} C_VEL
LIN {X 0,Y 195.283,Z 381.76,A -85,B 0,C 180,E1 -21808.267,E2 -21808.267} C_VEL
LIN {X 0,Y 196.993,Z 382.963,A -85,B 0,C 180,E1 -21809.315,E2 -21809.315} C_VEL
LIN {X 0,Y 198.616,Z 386.045,A -85,B 0,C 180,E1 -21810.501,E2 -21810.501} C_VEL
LIN {X 0,Y 201.086,Z 388.601,A -85,B 0,C 180,E1 -21811.972,E2 -21811.972} C_VEL
LIN {X 0,Y 203.366,Z 392.063,A -85,B 0,C 180,E1 -21813.42,E2 -21813.42} C_VEL
LIN {X 0,Y 204.424,Z 393.368,A -85,B 0,C 180,E1 -21814.039,E2 -21814.039} C_VEL
LIN {X 0,Y 207.113,Z 397.29,A -85,B 0,C 180,E1 -21815.624,E2 -21815.624} C_VEL
LIN {X 0,Y 211.913,Z 405.266,A -85,B 0,C 180,E1 -21818.513,E2 -21818.513} C_VEL
LIN {X 0,Y 216.374,Z 413.966,A -85,B 0,C 180,E1 -21821.313,E2 -21821.313} C_VEL
LIN {X 0,Y 219.33,Z 422.06,A -85,B 0,C 180,E1 -21823.546,E2 -21823.546} C_VEL
LIN {X 0,Y 221.944,Z 432.016,A -85,B 0,C 180,E1 -21826.087,E2 -21826.087} C_VEL
LIN {X 0,Y 223.705,Z 442.537,A -85,B 0,C 180,E1 -21828.719,E2 -21828.719} C_VEL
LIN {X 0,Y 224.111,Z 448.276,A -85,B 0,C 180,E1 -21830.119,E2 -21830.119} C_VEL
LIN {X 0,Y 219.709,Z 460.533,A -85,B 0,C 180,E1 -21832.282,E2 -21832.282} C_VEL
LIN {X 0,Y 215.135,Z 471.409,A -85,B 0,C 180,E1 -21834.612,E2 -21834.612} C_VEL
LIN {X 0,Y 210.936,Z 481.128,A -85,B 0,C 180,E1 -21837.219,E2 -21837.219} C_VEL
LIN {X 0,Y 206.292,Z 490.78,A -85,B 0,C 180,E1 -21840.396,E2 -21840.396} C_VEL
LIN {X 0,Y 202.241,Z 498.816,A -85,B 0,C 180,E1 -21843.699,E2 -21843.699} C_VEL
LIN {X 0,Y 198.785,Z 505.44,A -85,B 0,C 180,E1 -21847.113,E2 -21847.113} C_VEL
LIN {X 0,Y 195.702,Z 511.555,A -85,B 0,C 180,E1 -21851.142,E2 -21851.142} C_VEL
LIN {X 0,Y 193.409,Z 516.267,A -85,B 0,C 180,E1 -21855.263,E2 -21855.263} C_VEL
LIN {X 0,Y 191.805,Z 519.711,A -85,B 0,C 180,E1 -21859.442,E2 -21859.442} C_VEL
LIN {X 0,Y 190.945,Z 521.977,A -85,B 0,C 180,E1 -21863.66,E2 -21863.66} C_VEL
LIN {X 0,Y 190.605,Z 523.126,A -85,B 0,C 180,E1 -21867.886,E2 -21867.886} C_VEL
LIN {X 0,Y 190.602,Z 523.138,A -85,B 0,C 180,E1 -21872.112,E2 -21872.112} C_VEL
LIN {X 0,Y 190.924,Z 522.036,A -85,B 0,C 180,E1 -21876.339,E2 -21876.339} C_VEL
LIN {X 0,Y 191.799,Z 519.814,A -85,B 0,C 180,E1 -21880.556,E2 -21880.556} C_VEL
LIN {X 0,Y 193.34,Z 516.413,A -85,B 0,C 180,E1 -21884.74,E2 -21884.74} C_VEL
LIN {X 0,Y 195.654,Z 511.745,A -85,B 0,C 180,E1 -21888.861,E2 -21888.861} C_VEL
LIN {X 0,Y 198.696,Z 505.69,A -85,B 0,C 180,E1 -21892.896,E2 -21892.896} C_VEL
LIN {X 0,Y 202.711,Z 498.044,A -85,B 0,C 180,E1 -21896.788,E2 -21896.788} C_VEL
LIN {X 0,Y 206.838,Z 489.885,A -85,B 0,C 180,E1 -21900.077,E2 -21900.077} C_VEL
LIN {X 0,Y 211.563,Z 480.043,A -85,B 0,C 180,E1 -21903.237,E2 -21903.237} C_VEL
LIN {X 0,Y 215.89,Z 469.956,A -85,B 0,C 180,E1 -21905.87,E2 -21905.87} C_VEL
LIN {X 0,Y 220.457,Z 458.975,A -85,B 0,C 180,E1 -21908.144,E2 -21908.144} C_VEL
LIN {X 0,Y 224.114,Z 448.723,A -85,B 0,C 180,E1 -21909.932,E2 -21909.932} C_VEL
LIN {X 0,Y 224.036,Z 445.033,A -85,B 0,C 180,E1 -21910.817,E2 -21910.817} C_VEL
LIN {X 0,Y 222.524,Z 434.549,A -85,B 0,C 180,E1 -21913.413,E2 -21913.413} C_VEL
LIN {X 0,Y 220.134,Z 424.378,A -85,B 0,C 180,E1 -21916.003,E2 -21916.003} C_VEL
LIN {X 0,Y 217.195,Z 415.791,A -85,B 0,C 180,E1 -21918.321,E2 -21918.321} C_VEL
LIN {X 0,Y 213.525,Z 408.194,A -85,B 0,C 180,E1 -21920.684,E2 -21920.684} C_VEL
LIN {X 0,Y 209.248,Z 400.883,A -85,B 0,C 180,E1 -21923.254,E2 -21923.254} C_VEL
LIN {X 0,Y 206.561,Z 396.651,A -85,B 0,C 180,E1 -21924.885,E2 -21924.885} C_VEL
LIN {X 0,Y 203.648,Z 392.358,A -85,B 0,C 180,E1 -21926.632,E2 -21926.632} C_VEL
LIN {X 0,Y 201.276,Z 388.991,A -85,B 0,C 180,E1 -21928.121,E2 -21928.121} C_VEL
LIN {X 0,Y 200.357,Z 387.678,A -85,B 0,C 180,E1 -21928.695,E2 -21928.695} C_VEL
LIN {X 0,Y 198.115,Z 385.262,A -85,B 0,C 180,E1 -21930.075,E2 -21930.075} C_VEL
LIN {X 0,Y 196.866,Z 382.734,A -85,B 0,C 180,E1 -21931.021,E2 -21931.021} C_VEL
LIN {X 0,Y 194.325,Z 380.861,A -85,B 0,C 180,E1 -21932.613,E2 -21932.613} C_VEL
LIN {X 0,Y 192.957,Z 378.577,A -85,B 0,C 180,E1 -21933.647,E2 -21933.647} C_VEL
LIN {X 0,Y 192.601,Z 377.093,A -85,B 0,C 180,E1 -21934.031,E2 -21934.031} C_VEL
LIN {X 0,Y 192.704,Z 377.105,A -85,B 0,C 180,E1 -21936.348,E2 -21936.348} C_VEL
LIN {X 0,Y 192.73,Z 377.08,A -85,B 0,C 180,E1 -21941.457,E2 -21941.457} C_VEL
LIN {X 0,Y 192.763,Z 377.07,A -85,B 0,C 180,E1 -21945.213,E2 -21945.213} C_VEL
LIN {X 0,Y 193.018,Z 377.053,A -85,B 0,C 180,E1 -21949.51,E2 -21949.51} C_VEL
LIN {X 0,Y 193.004,Z 377.068,A -85,B 0,C 180,E1 -21953.728,E2 -21953.728} C_VEL
LIN {X 0,Y 193.263,Z 377.037,A -85,B 0,C 180,E1 -21957.916,E2 -21957.916} C_VEL
LIN {X 0,Y 193.445,Z 377.015,A -85,B 0,C 180,E1 -21960,E2 -21960} C_VEL
LIN {X 0,Y 192.979,Z 377.073,A -85,B 0,C 180,E1 -21964.177,E2 -21964.177} C_VEL
LIN {X 0,Y 193.077,Z 377.059,A -85,B 0,C 180,E1 -21968.372,E2 -21968.372} C_VEL
LIN {X 0,Y 193.008,Z 377.068,A -85,B 0,C 180,E1 -21970.538,E2 -21970.538} C_VEL
LIN {X 0,Y 192.821,Z 377.083,A -85,B 0,C 180,E1 -21972.632,E2 -21972.632} C_VEL
LIN {X 0,Y 192.987,Z 378.531,A -85,B 0,C 180,E1 -21976.938,E2 -21976.938} C_VEL
LIN {X 0,Y 193.147,Z 380.263,A -85,B 0,C 180,E1 -21981.338,E2 -21981.338} C_VEL
LIN {X 0,Y 193.501,Z 382.435,A -85,B 0,C 180,E1 -21986.128,E2 -21986.128} C_VEL
LIN {X 0,Y 193.608,Z 382.883,A -85,B 0,C 180,E1 -21986.402,E2 -21986.402} C_VEL
LIN {X 0,Y 194.76,Z 385.777,A -85,B 0,C 180,E1 -21987.32,E2 -21987.32} C_VEL
LIN {X 0,Y 197.035,Z 388.623,A -85,B 0,C 180,E1 -21988.803,E2 -21988.803} C_VEL
LIN {X 0,Y 198.02,Z 389.649,A -85,B 0,C 180,E1 -21989.397,E2 -21989.397} C_VEL
LIN {X 0,Y 199.697,Z 393.13,A -85,B 0,C 180,E1 -21990.537,E2 -21990.537} C_VEL
LIN {X 0,Y 201.968,Z 396.182,A -85,B 0,C 180,E1 -21991.903,E2 -21991.903} C_VEL
LIN {X 0,Y 204.177,Z 400.287,A -85,B 0,C 180,E1 -21993.27,E2 -21993.27} C_VEL
LIN {X 0,Y 205.413,Z 402.198,A -85,B 0,C 180,E1 -21993.999,E2 -21993.999} C_VEL
LIN {X 0,Y 207.9,Z 406.755,A -85,B 0,C 180,E1 -21995.493,E2 -21995.493} C_VEL
LIN {X 0,Y 211.456,Z 414.394,A -85,B 0,C 180,E1 -21997.716,E2 -21997.716} C_VEL
LIN {X 0,Y 215.235,Z 423.371,A -85,B 0,C 180,E1 -22000.157,E2 -22000.157} C_VEL
LIN {X 0,Y 217.325,Z 431.182,A -85,B 0,C 180,E1 -22001.946,E2 -22001.946} C_VEL
LIN {X 0,Y 219.25,Z 443.936,A -85,B 0,C 180,E1 -22004.635,E2 -22004.635} C_VEL
LIN {X 0,Y 219.953,Z 456.669,A -85,B 0,C 180,E1 -22007.299,E2 -22007.299} C_VEL
LIN {X 0,Y 219.512,Z 468.642,A -85,B 0,C 180,E1 -22009.886,E2 -22009.886} C_VEL
LIN {X 0,Y 218.817,Z 473.902,A -85,B 0,C 180,E1 -22011.043,E2 -22011.043} C_VEL
LIN {X 0,Y 214.209,Z 484.905,A -85,B 0,C 180,E1 -22013.22,E2 -22013.22} C_VEL
LIN {X 0,Y 209.546,Z 495.464,A -85,B 0,C 180,E1 -22015.822,E2 -22015.822} C_VEL
LIN {X 0,Y 204.775,Z 505.808,A -85,B 0,C 180,E1 -22019.016,E2 -22019.016} C_VEL
LIN {X 0,Y 200.755,Z 514.425,A -85,B 0,C 180,E1 -22022.365,E2 -22022.365} C_VEL
LIN {X 0,Y 197.184,Z 521.597,A -85,B 0,C 180,E1 -22025.804,E2 -22025.804} C_VEL
LIN {X 0,Y 194.205,Z 528.28,A -85,B 0,C 180,E1 -22029.894,E2 -22029.894} C_VEL
LIN {X 0,Y 192.798,Z 531.591,A -85,B 0,C 180,E1 -22032.403,E2 -22032.403} C_VEL
LIN {X 0,Y 191.391,Z 533.503,A -85,B 0,C 180,E1 -22034.018,E2 -22034.018} C_VEL
LIN {X 0,Y 187.606,Z 536.162,A -85,B 0,C 180,E1 -22036.668,E2 -22036.668} C_VEL
LIN {X 0,Y 184.683,Z 537.882,A -85,B 0,C 180,E1 -22038.885,E2 -22038.885} C_VEL
LIN {X 0,Y 183.395,Z 538.934,A -85,B 0,C 180,E1 -22040.656,E2 -22040.656} C_VEL
LIN {X 0,Y 183.255,Z 539.236,A -85,B 0,C 180,E1 -22041.264,E2 -22041.264} C_VEL
LIN {X 0,Y 183.227,Z 541.028,A -85,B 0,C 180,E1 -22045.769,E2 -22045.769} C_VEL
LIN {X 0,Y 183.414,Z 541.611,A -85,B 0,C 180,E1 -22050.001,E2 -22050.001} C_VEL
LIN {X 0,Y 183.232,Z 540.975,A -85,B 0,C 180,E1 -22054.4,E2 -22054.4} C_VEL
LIN {X 0,Y 183.286,Z 539.161,A -85,B 0,C 180,E1 -22058.824,E2 -22058.824} C_VEL
LIN {X 0,Y 183.997,Z 536.162,A -85,B 0,C 180,E1 -22063.25,E2 -22063.25} C_VEL
LIN {X 0,Y 185.658,Z 531.924,A -85,B 0,C 180,E1 -22067.629,E2 -22067.629} C_VEL
LIN {X 0,Y 188.174,Z 526.33,A -85,B 0,C 180,E1 -22071.932,E2 -22071.932} C_VEL
LIN {X 0,Y 191.621,Z 519.238,A -85,B 0,C 180,E1 -22076.112,E2 -22076.112} C_VEL
LIN {X 0,Y 195.52,Z 511.676,A -85,B 0,C 180,E1 -22079.621,E2 -22079.621} C_VEL
LIN {X 0,Y 199.996,Z 502.568,A -85,B 0,C 180,E1 -22083.004,E2 -22083.004} C_VEL
LIN {X 0,Y 205.256,Z 491.643,A -85,B 0,C 180,E1 -22086.204,E2 -22086.204} C_VEL
LIN {X 0,Y 210.309,Z 480.411,A -85,B 0,C 180,E1 -22088.799,E2 -22088.799} C_VEL
LIN {X 0,Y 212.499,Z 475.258,A -85,B 0,C 180,E1 -22089.799,E2 -22089.799} C_VEL
LIN {X 0,Y 213.258,Z 471.195,A -85,B 0,C 180,E1 -22090.715,E2 -22090.715} C_VEL
LIN {X 0,Y 213.9,Z 461.605,A -85,B 0,C 180,E1 -22092.94,E2 -22092.94} C_VEL
LIN {X 0,Y 213.833,Z 450.33,A -85,B 0,C 180,E1 -22095.425,E2 -22095.425} C_VEL
LIN {X 0,Y 212.776,Z 438.969,A -85,B 0,C 180,E1 -22097.941,E2 -22097.941} C_VEL
LIN {X 0,Y 211.14,Z 430.154,A -85,B 0,C 180,E1 -22099.959,E2 -22099.959} C_VEL
LIN {X 0,Y 208.541,Z 422.41,A -85,B 0,C 180,E1 -22102.045,E2 -22102.045} C_VEL
LIN {X 0,Y 203.83,Z 411.721,A -85,B 0,C 180,E1 -22105.326,E2 -22105.326} C_VEL
LIN {X 0,Y 201.116,Z 406.39,A -85,B 0,C 180,E1 -22107.167,E2 -22107.167} C_VEL
LIN {X 0,Y 198.745,Z 401.995,A -85,B 0,C 180,E1 -22108.784,E2 -22108.784} C_VEL
LIN {X 0,Y 195.713,Z 397.087,A -85,B 0,C 180,E1 -22110.855,E2 -22110.855} C_VEL
LIN {X 0,Y 194.755,Z 395.108,A -85,B 0,C 180,E1 -22111.583,E2 -22111.583} C_VEL
LIN {X 0,Y 192.225,Z 391.754,A -85,B 0,C 180,E1 -22113.393,E2 -22113.393} C_VEL
LIN {X 0,Y 190.879,Z 388.817,A -85,B 0,C 180,E1 -22114.499,E2 -22114.499} C_VEL
LIN {X 0,Y 187.796,Z 385.603,A -85,B 0,C 180,E1 -22116.862,E2 -22116.862} C_VEL
LIN {X 0,Y 186.393,Z 382.63,A -85,B 0,C 180,E1 -22118.213,E2 -22118.213} C_VEL
LIN {X 0,Y 186.201,Z 381.715,A -85,B 0,C 180,E1 -22118.553,E2 -22118.553} C_VEL
LIN {X 0,Y 186.043,Z 380.201,A -85,B 0,C 180,E1 -22122.41,E2 -22122.41} C_VEL
LIN {X 0,Y 185.895,Z 378.703,A -85,B 0,C 180,E1 -22126.889,E2 -22126.889} C_VEL
LIN {X 0,Y 185.947,Z 377.955,A -85,B 0,C 180,E1 -22129.327,E2 -22129.327} C_VEL
LIN {X 0,Y 185.973,Z 377.942,A -85,B 0,C 180,E1 -22133.491,E2 -22133.491} C_VEL
LIN {X 0,Y 186.213,Z 377.914,A -85,B 0,C 180,E1 -22137.837,E2 -22137.837} C_VEL
LIN {X 0,Y 186.411,Z 377.884,A -85,B 0,C 180,E1 -22140,E2 -22140} C_VEL
LIN {X 0,Y 185.932,Z 377.946,A -85,B 0,C 180,E1 -22144.336,E2 -22144.336} C_VEL
LIN {X 0,Y 186.033,Z 377.938,A -85,B 0,C 180,E1 -22148.692,E2 -22148.692} C_VEL
LIN {X 0,Y 185.739,Z 377.931,A -85,B 0,C 180,E1 -22153.122,E2 -22153.122} C_VEL
LIN {X 0,Y 185.693,Z 377.968,A -85,B 0,C 180,E1 -22157.625,E2 -22157.625} C_VEL
LIN {X 0,Y 185.587,Z 377.976,A -85,B 0,C 180,E1 -22161.449,E2 -22161.449} C_VEL
LIN {X 0,Y 186.187,Z 380.049,A -85,B 0,C 180,E1 -22162.177,E2 -22162.177} C_VEL
LIN {X 0,Y 187.743,Z 382.205,A -85,B 0,C 180,E1 -22163.583,E2 -22163.583} C_VEL
LIN {X 0,Y 190.267,Z 383.909,A -85,B 0,C 180,E1 -22165.503,E2 -22165.503} C_VEL
LIN {X 0,Y 191.587,Z 386.68,A -85,B 0,C 180,E1 -22166.703,E2 -22166.703} C_VEL
LIN {X 0,Y 194.429,Z 389.516,A -85,B 0,C 180,E1 -22168.704,E2 -22168.704} C_VEL
LIN {X 0,Y 196.218,Z 392.646,A -85,B 0,C 180,E1 -22170.096,E2 -22170.096} C_VEL
LIN {X 0,Y 198.011,Z 394.599,A -85,B 0,C 180,E1 -22171.271,E2 -22171.271} C_VEL
LIN {X 0,Y 200.385,Z 398.212,A -85,B 0,C 180,E1 -22172.893,E2 -22172.893} C_VEL
LIN {X 0,Y 204.614,Z 405.025,A -85,B 0,C 180,E1 -22175.726,E2 -22175.726} C_VEL
LIN {X 0,Y 208.111,Z 411.15,A -85,B 0,C 180,E1 -22178.047,E2 -22178.047} C_VEL
LIN {X 0,Y 211.345,Z 417.705,A -85,B 0,C 180,E1 -22180.3,E2 -22180.3} C_VEL
LIN {X 0,Y 214.159,Z 425.662,A -85,B 0,C 180,E1 -22182.661,E2 -22182.661} C_VEL
LIN {X 0,Y 216.366,Z 434.959,A -85,B 0,C 180,E1 -22185.194,E2 -22185.194} C_VEL
LIN {X 0,Y 217.912,Z 445.197,A -85,B 0,C 180,E1 -22187.884,E2 -22187.884} C_VEL
LIN {X 0,Y 218.124,Z 450.372,A -85,B 0,C 180,E1 -22189.208,E2 -22189.208} C_VEL
LIN {X 0,Y 213.703,Z 461.946,A -85,B 0,C 180,E1 -22191.328,E2 -22191.328} C_VEL
LIN {X 0,Y 208.907,Z 472.826,A -85,B 0,C 180,E1 -22193.751,E2 -22193.751} C_VEL
LIN {X 0,Y 204.251,Z 482.95,A -85,B 0,C 180,E1 -22196.595,E2 -22196.595} C_VEL
LIN {X 0,Y 199.497,Z 492.347,A -85,B 0,C 180,E1 -22199.866,E2 -22199.866} C_VEL
LIN {X 0,Y 195.322,Z 500.162,A -85,B 0,C 180,E1 -22203.27,E2 -22203.27} C_VEL
LIN {X 0,Y 191.391,Z 507.443,A -85,B 0,C 180,E1 -22207.32,E2 -22207.32} C_VEL
LIN {X 0,Y 188.266,Z 513.211,A -85,B 0,C 180,E1 -22211.499,E2 -22211.499} C_VEL
LIN {X 0,Y 186.516,Z 516.617,A -85,B 0,C 180,E1 -22214.706,E2 -22214.706} C_VEL
LIN {X 0,Y 184.821,Z 520.06,A -85,B 0,C 180,E1 -22219.039,E2 -22219.039} C_VEL
LIN {X 0,Y 183.883,Z 522.381,A -85,B 0,C 180,E1 -22223.577,E2 -22223.577} C_VEL
LIN {X 0,Y 183.526,Z 523.474,A -85,B 0,C 180,E1 -22227.804,E2 -22227.804} C_VEL
LIN {X 0,Y 183.523,Z 523.485,A -85,B 0,C 180,E1 -22232.194,E2 -22232.194} C_VEL
LIN {X 0,Y 183.861,Z 522.384,A -85,B 0,C 180,E1 -22236.584,E2 -22236.584} C_VEL
LIN {X 0,Y 184.815,Z 520.162,A -85,B 0,C 180,E1 -22240.96,E2 -22240.96} C_VEL
LIN {X 0,Y 186.453,Z 516.761,A -85,B 0,C 180,E1 -22245.298,E2 -22245.298} C_VEL
LIN {X 0,Y 188.949,Z 512.092,A -85,B 0,C 180,E1 -22249.557,E2 -22249.557} C_VEL
LIN {X 0,Y 192.143,Z 506.039,A -85,B 0,C 180,E1 -22253.724,E2 -22253.724} C_VEL
LIN {X 0,Y 196.391,Z 498.391,A -85,B 0,C 180,E1 -22257.723,E2 -22257.723} C_VEL
LIN {X 0,Y 200.718,Z 490.232,A -85,B 0,C 180,E1 -22261.094,E2 -22261.094} C_VEL
LIN {X 0,Y 205.652,Z 480.389,A -85,B 0,C 180,E1 -22264.323,E2 -22264.323} C_VEL
LIN {X 0,Y 210.164,Z 470.302,A -85,B 0,C 180,E1 -22267.007,E2 -22267.007} C_VEL
LIN {X 0,Y 214.932,Z 459.318,A -85,B 0,C 180,E1 -22269.31,E2 -22269.31} C_VEL
LIN {X 0,Y 218.06,Z 450.898,A -85,B 0,C 180,E1 -22270.84,E2 -22270.84} C_VEL
LIN {X 0,Y 218.19,Z 448.046,A -85,B 0,C 180,E1 -22271.505,E2 -22271.505} C_VEL
LIN {X 0,Y 216.994,Z 437.846,A -85,B 0,C 180,E1 -22274.193,E2 -22274.193} C_VEL
LIN {X 0,Y 215.03,Z 428.652,A -85,B 0,C 180,E1 -22276.657,E2 -22276.657} C_VEL
LIN {X 0,Y 212.897,Z 421.486,A -85,B 0,C 180,E1 -22278.683,E2 -22278.683} C_VEL
LIN {X 0,Y 210.363,Z 415.467,A -85,B 0,C 180,E1 -22280.597,E2 -22280.597} C_VEL
LIN {X 0,Y 206.241,Z 407.717,A -85,B 0,C 180,E1 -22283.391,E2 -22283.391} C_VEL
LIN {X 0,Y 202.469,Z 401.567,A -85,B 0,C 180,E1 -22285.888,E2 -22285.888} C_VEL
LIN {X 0,Y 200.516,Z 398.361,A -85,B 0,C 180,E1 -22287.242,E2 -22287.242} C_VEL
LIN {X 0,Y 198.097,Z 394.762,A -85,B 0,C 180,E1 -22288.893,E2 -22288.893} C_VEL
LIN {X 0,Y 197.039,Z 393.484,A -85,B 0,C 180,E1 -22289.599,E2 -22289.599} C_VEL
LIN {X 0,Y 194.818,Z 390.352,A -85,B 0,C 180,E1 -22291.225,E2 -22291.225} C_VEL
LIN {X 0,Y 194.116,Z 389.051,A -85,B 0,C 180,E1 -22291.775,E2 -22291.775} C_VEL
LIN {X 0,Y 191.637,Z 386.738,A -85,B 0,C 180,E1 -22293.524,E2 -22293.524} C_VEL
LIN {X 0,Y 190.183,Z 383.757,A -85,B 0,C 180,E1 -22294.851,E2 -22294.851} C_VEL
LIN {X 0,Y 187.448,Z 381.924,A -85,B 0,C 180,E1 -22296.962,E2 -22296.962} C_VEL
LIN {X 0,Y 186.025,Z 379.679,A -85,B 0,C 180,E1 -22298.313,E2 -22298.313} C_VEL
LIN {X 0,Y 185.594,Z 377.957,A -85,B 0,C 180,E1 -22298.915,E2 -22298.915} C_VEL
LIN {X 0,Y 185.689,Z 377.971,A -85,B 0,C 180,E1 -22302.375,E2 -22302.375} C_VEL
LIN {X 0,Y 185.733,Z 377.935,A -85,B 0,C 180,E1 -22306.877,E2 -22306.877} C_VEL
LIN {X 0,Y 186.028,Z 377.937,A -85,B 0,C 180,E1 -22311.308,E2 -22311.308} C_VEL
LIN {X 0,Y 186.207,Z 377.916,A -85,B 0,C 180,E1 -22317.837,E2 -22317.837} C_VEL
LIN {X 0,Y 186.408,Z 377.891,A -85,B 0,C 180,E1 -22320,E2 -22320} C_VEL
LIN {X 0,Y 185.927,Z 377.951,A -85,B 0,C 180,E1 -22324.335,E2 -22324.335} C_VEL
LIN {X 0,Y 186.027,Z 377.938,A -85,B 0,C 180,E1 -22328.691,E2 -22328.691} C_VEL
LIN {X 0,Y 185.936,Z 378.077,A -85,B 0,C 180,E1 -22330.894,E2 -22330.894} C_VEL
LIN {X 0,Y 185.964,Z 379.478,A -85,B 0,C 180,E1 -22335.34,E2 -22335.34} C_VEL
LIN {X 0,Y 186.108,Z 381.116,A -85,B 0,C 180,E1 -22339.869,E2 -22339.869} C_VEL
LIN {X 0,Y 186.241,Z 381.856,A -85,B 0,C 180,E1 -22341.37,E2 -22341.37} C_VEL
LIN {X 0,Y 187.164,Z 384.428,A -85,B 0,C 180,E1 -22342.345,E2 -22342.345} C_VEL
LIN {X 0,Y 189.629,Z 387.618,A -85,B 0,C 180,E1 -22344.399,E2 -22344.399} C_VEL
LIN {X 0,Y 191.089,Z 389.096,A -85,B 0,C 180,E1 -22345.48,E2 -22345.48} C_VEL
LIN {X 0,Y 193.037,Z 393.065,A -85,B 0,C 180,E1 -22347.071,E2 -22347.071} C_VEL
LIN {X 0,Y 195.189,Z 395.727,A -85,B 0,C 180,E1 -22348.568,E2 -22348.568} C_VEL
LIN {X 0,Y 197.248,Z 399.708,A -85,B 0,C 180,E1 -22350.069,E2 -22350.069} C_VEL
LIN {X 0,Y 198.745,Z 401.865,A -85,B 0,C 180,E1 -22351.068,E2 -22351.068} C_VEL
LIN {X 0,Y 200.96,Z 406.168,A -85,B 0,C 180,E1 -22352.616,E2 -22352.616} C_VEL
LIN {X 0,Y 202.071,Z 408.157,A -85,B 0,C 180,E1 -22353.341,E2 -22353.341} C_VEL
LIN {X 0,Y 206.052,Z 416.359,A -85,B 0,C 180,E1 -22356.056,E2 -22356.056} C_VEL
LIN {X 0,Y 209.92,Z 425.991,A -85,B 0,C 180,E1 -22358.883,E2 -22358.883} C_VEL
LIN {X 0,Y 211.931,Z 433.466,A -85,B 0,C 180,E1 -22360.756,E2 -22360.756} C_VEL
LIN {X 0,Y 213.527,Z 444.716,A -85,B 0,C 180,E1 -22363.282,E2 -22363.282} C_VEL
LIN {X 0,Y 214.078,Z 456.81,A -85,B 0,C 180,E1 -22365.949,E2 -22365.949} C_VEL
LIN {X 0,Y 213.508,Z 469.468,A -85,B 0,C 180,E1 -22368.828,E2 -22368.828} C_VEL
LIN {X 0,Y 213.078,Z 473.554,A -85,B 0,C 180,E1 -22369.787,E2 -22369.787} C_VEL
LIN {X 0,Y 211.204,Z 478.54,A -85,B 0,C 180,E1 -22370.785,E2 -22370.785} C_VEL
LIN {X 0,Y 206.06,Z 490.064,A -85,B 0,C 180,E1 -22373.355,E2 -22373.355} C_VEL
LIN {X 0,Y 201.388,Z 499.774,A -85,B 0,C 180,E1 -22376.058,E2 -22376.058} C_VEL
LIN {X 0,Y 197.065,Z 508.686,A -85,B 0,C 180,E1 -22379.147,E2 -22379.147} C_VEL
LIN {X 0,Y 192.719,Z 517.315,A -85,B 0,C 180,E1 -22382.882,E2 -22382.882} C_VEL
LIN {X 0,Y 188.947,Z 524.777,A -85,B 0,C 180,E1 -22387.012,E2 -22387.012} C_VEL
LIN {X 0,Y 186.199,Z 530.717,A -85,B 0,C 180,E1 -22391.288,E2 -22391.288} C_VEL
LIN {X 0,Y 184.739,Z 534.262,A -85,B 0,C 180,E1 -22394.557,E2 -22394.557} C_VEL
LIN {X 0,Y 183.536,Z 537.855,A -85,B 0,C 180,E1 -22398.963,E2 -22398.963} C_VEL
LIN {X 0,Y 183.255,Z 539.236,A -85,B 0,C 180,E1 -22401.264,E2 -22401.264} C_VEL
LIN {X 0,Y 182.513,Z 540.104,A -85,B 0,C 180,E1 -22403.084,E2 -22403.084} C_VEL
LIN {X 0,Y 180.967,Z 540.714,A -85,B 0,C 180,E1 -22404.883,E2 -22404.883} C_VEL
LIN {X 0,Y 177.393,Z 541.233,A -85,B 0,C 180,E1 -22408.543,E2 -22408.543} C_VEL
LIN {X 0,Y 176.219,Z 541.182,A -85,B 0,C 180,E1 -22411.105,E2 -22411.105} C_VEL
LIN {X 0,Y 176.144,Z 540.627,A -85,B 0,C 180,E1 -22414.578,E2 -22414.578} C_VEL
LIN {X 0,Y 176.226,Z 538.81,A -85,B 0,C 180,E1 -22419.18,E2 -22419.18} C_VEL
LIN {X 0,Y 177.022,Z 535.81,A -85,B 0,C 180,E1 -22423.782,E2 -22423.782} C_VEL
LIN {X 0,Y 178.836,Z 531.571,A -85,B 0,C 180,E1 -22428.325,E2 -22428.325} C_VEL
LIN {X 0,Y 181.516,Z 525.976,A -85,B 0,C 180,E1 -22432.78,E2 -22432.78} C_VEL
LIN {X 0,Y 185.207,Z 518.884,A -85,B 0,C 180,E1 -22437.089,E2 -22437.089} C_VEL
LIN {X 0,Y 189.324,Z 511.323,A -85,B 0,C 180,E1 -22440.693,E2 -22440.693} C_VEL
LIN {X 0,Y 194.008,Z 502.214,A -85,B 0,C 180,E1 -22444.16,E2 -22444.16} C_VEL
LIN {X 0,Y 199.518,Z 491.289,A -85,B 0,C 180,E1 -22447.419,E2 -22447.419} C_VEL
LIN {X 0,Y 204.798,Z 480.059,A -85,B 0,C 180,E1 -22450.05,E2 -22450.05} C_VEL
LIN {X 0,Y 206.696,Z 475.521,A -85,B 0,C 180,E1 -22450.966,E2 -22450.966} C_VEL
LIN {X 0,Y 207.813,Z 467.039,A -85,B 0,C 180,E1 -22453.046,E2 -22453.046} C_VEL
LIN {X 0,Y 208.194,Z 455.403,A -85,B 0,C 180,E1 -22455.796,E2 -22455.796} C_VEL
LIN {X 0,Y 207.764,Z 445.567,A -85,B 0,C 180,E1 -22458.091,E2 -22458.091} C_VEL
LIN {X 0,Y 206.562,Z 435.962,A -85,B 0,C 180,E1 -22460.362,E2 -22460.362} C_VEL
LIN {X 0,Y 204.931,Z 429.661,A -85,B 0,C 180,E1 -22462.072,E2 -22462.072} C_VEL
LIN {X 0,Y 201.499,Z 420.747,A -85,B 0,C 180,E1 -22464.866,E2 -22464.866} C_VEL
LIN {X 0,Y 197.498,Z 411.874,A -85,B 0,C 180,E1 -22467.965,E2 -22467.965} C_VEL
LIN {X 0,Y 194.786,Z 406.591,A -85,B 0,C 180,E1 -22470.063,E2 -22470.063} C_VEL
LIN {X 0,Y 192.451,Z 402.349,A -85,B 0,C 180,E1 -22471.881,E2 -22471.881} C_VEL
LIN {X 0,Y 191.709,Z 400.907,A -85,B 0,C 180,E1 -22472.504,E2 -22472.504} C_VEL
LIN {X 0,Y 189.383,Z 397.364,A -85,B 0,C 180,E1 -22474.37,E2 -22474.37} C_VEL
LIN {X 0,Y 188.36,Z 395.032,A -85,B 0,C 180,E1 -22475.328,E2 -22475.328} C_VEL
LIN {X 0,Y 185.614,Z 391.813,A -85,B 0,C 180,E1 -22477.678,E2 -22477.678} C_VEL
LIN {X 0,Y 183.813,Z 388.029,A -85,B 0,C 180,E1 -22479.581,E2 -22479.581} C_VEL
LIN {X 0,Y 180.657,Z 384.723,A -85,B 0,C 180,E1 -22482.891,E2 -22482.891} C_VEL
LIN {X 0,Y 179.171,Z 381.472,A -85,B 0,C 180,E1 -22485.011,E2 -22485.011} C_VEL
LIN {X 0,Y 178.978,Z 380.662,A -85,B 0,C 180,E1 -22485.503,E2 -22485.503} C_VEL
LIN {X 0,Y 179.022,Z 379.604,A -85,B 0,C 180,E1 -22488.949,E2 -22488.949} C_VEL
LIN {X 0,Y 179,Z 379.059,A -85,B 0,C 180,E1 -22490.965,E2 -22490.965} C_VEL
LIN {X 0,Y 178.881,Z 378.828,A -85,B 0,C 180,E1 -22495.493,E2 -22495.493} C_VEL
LIN {X 0,Y 179.374,Z 378.76,A -85,B 0,C 180,E1 -22500,E2 -22500} C_VEL
LIN {X 0,Y 178.881,Z 378.826,A -85,B 0,C 180,E1 -22504.507,E2 -22504.507} C_VEL
LIN {X 0,Y 178.982,Z 378.816,A -85,B 0,C 180,E1 -22509.037,E2 -22509.037} C_VEL
LIN {X 0,Y 178.686,Z 379.026,A -85,B 0,C 180,E1 -22514.813,E2 -22514.813} C_VEL
LIN {X 0,Y 179.486,Z 381.461,A -85,B 0,C 180,E1 -22516.2,E2 -22516.2} C_VEL
LIN {X 0,Y 181.772,Z 383.882,A -85,B 0,C 180,E1 -22518.932,E2 -22518.932} C_VEL
LIN {X 0,Y 183.532,Z 384.851,A -85,B 0,C 180,E1 -22520.672,E2 -22520.672} C_VEL
LIN {X 0,Y 184.822,Z 387.699,A -85,B 0,C 180,E1 -22522.203,E2 -22522.203} C_VEL
LIN {X 0,Y 187.286,Z 390.079,A -85,B 0,C 180,E1 -22524.38,E2 -22524.38} C_VEL
LIN {X 0,Y 187.93,Z 390.681,A -85,B 0,C 180,E1 -22524.907,E2 -22524.907} C_VEL
LIN {X 0,Y 189.819,Z 393.936,A -85,B 0,C 180,E1 -22526.675,E2 -22526.675} C_VEL
LIN {X 0,Y 191.661,Z 395.941,A -85,B 0,C 180,E1 -22528.097,E2 -22528.097} C_VEL
LIN {X 0,Y 193.817,Z 399.361,A -85,B 0,C 180,E1 -22529.847,E2 -22529.847} C_VEL
LIN {X 0,Y 195.016,Z 400.911,A -85,B 0,C 180,E1 -22530.741,E2 -22530.741} C_VEL
LIN {X 0,Y 199.712,Z 408.522,A -85,B 0,C 180,E1 -22534.267,E2 -22534.267} C_VEL
LIN {X 0,Y 203.582,Z 415.716,A -85,B 0,C 180,E1 -22537.168,E2 -22537.168} C_VEL
LIN {X 0,Y 206.697,Z 422.418,A -85,B 0,C 180,E1 -22539.608,E2 -22539.608} C_VEL
LIN {X 0,Y 208.964,Z 429.366,A -85,B 0,C 180,E1 -22541.795,E2 -22541.795} C_VEL
LIN {X 0,Y 210.943,Z 438.424,A -85,B 0,C 180,E1 -22544.4,E2 -22544.4} C_VEL
LIN {X 0,Y 212.132,Z 448.219,A -85,B 0,C 180,E1 -22547.14,E2 -22547.14} C_VEL
LIN {X 0,Y 212.308,Z 452.112,A -85,B 0,C 180,E1 -22548.193,E2 -22548.193} C_VEL
LIN {X 0,Y 207.749,Z 463.359,A -85,B 0,C 180,E1 -22550.317,E2 -22550.317} C_VEL
LIN {X 0,Y 202.478,Z 474.776,A -85,B 0,C 180,E1 -22552.971,E2 -22552.971} C_VEL
LIN {X 0,Y 197.617,Z 484.771,A -85,B 0,C 180,E1 -22555.934,E2 -22555.934} C_VEL
LIN {X 0,Y 192.703,Z 493.914,A -85,B 0,C 180,E1 -22559.296,E2 -22559.296} C_VEL
LIN {X 0,Y 189.004,Z 500.511,A -85,B 0,C 180,E1 -22562.301,E2 -22562.301} C_VEL
LIN {X 0,Y 184.836,Z 507.794,A -85,B 0,C 180,E1 -22566.468,E2 -22566.468} C_VEL
LIN {X 0,Y 181.547,Z 513.56,A -85,B 0,C 180,E1 -22570.788,E2 -22570.788} C_VEL
LIN {X 0,Y 179.65,Z 516.968,A -85,B 0,C 180,E1 -22574.106,E2 -22574.106} C_VEL
LIN {X 0,Y 177.839,Z 520.41,A -85,B 0,C 180,E1 -22578.603,E2 -22578.603} C_VEL
LIN {X 0,Y 176.789,Z 522.838,A -85,B 0,C 180,E1 -22583.639,E2 -22583.639} C_VEL
LIN {X 0,Y 176.45,Z 523.821,A -85,B 0,C 180,E1 -22587.716,E2 -22587.716} C_VEL
LIN {X 0,Y 176.445,Z 523.832,A -85,B 0,C 180,E1 -22592.282,E2 -22592.282} C_VEL
LIN {X 0,Y 176.812,Z 522.732,A -85,B 0,C 180,E1 -22596.848,E2 -22596.848} C_VEL
LIN {X 0,Y 177.831,Z 520.51,A -85,B 0,C 180,E1 -22601.396,E2 -22601.396} C_VEL
LIN {X 0,Y 179.596,Z 517.109,A -85,B 0,C 180,E1 -22605.897,E2 -22605.897} C_VEL
LIN {X 0,Y 182.272,Z 512.439,A -85,B 0,C 180,E1 -22610.304,E2 -22610.304} C_VEL
LIN {X 0,Y 185.661,Z 506.385,A -85,B 0,C 180,E1 -22614.606,E2 -22614.606} C_VEL
LIN {X 0,Y 190.136,Z 498.737,A -85,B 0,C 180,E1 -22618.718,E2 -22618.718} C_VEL
LIN {X 0,Y 194.657,Z 490.578,A -85,B 0,C 180,E1 -22622.176,E2 -22622.176} C_VEL
LIN {X 0,Y 199.813,Z 480.736,A -85,B 0,C 180,E1 -22625.474,E2 -22625.474} C_VEL
LIN {X 0,Y 204.546,Z 470.647,A -85,B 0,C 180,E1 -22628.203,E2 -22628.203} C_VEL
LIN {X 0,Y 209.496,Z 459.662,A -85,B 0,C 180,E1 -22630.539,E2 -22630.539} C_VEL
LIN {X 0,Y 212.409,Z 451.935,A -85,B 0,C 180,E1 -22631.994,E2 -22631.994} C_VEL
LIN {X 0,Y 211.823,Z 444.065,A -85,B 0,C 180,E1 -22634.166,E2 -22634.166} C_VEL
LIN {X 0,Y 210.341,Z 434.818,A -85,B 0,C 180,E1 -22636.769,E2 -22636.769} C_VEL
LIN {X 0,Y 207.929,Z 425.523,A -85,B 0,C 180,E1 -22639.552,E2 -22639.552} C_VEL
LIN {X 0,Y 204.844,Z 418.167,A -85,B 0,C 180,E1 -22642.101,E2 -22642.101} C_VEL
LIN {X 0,Y 199.948,Z 408.883,A -85,B 0,C 180,E1 -22645.779,E2 -22645.779} C_VEL
LIN {X 0,Y 196.694,Z 403.677,A -85,B 0,C 180,E1 -22648.195,E2 -22648.195} C_VEL
LIN {X 0,Y 194.482,Z 400.037,A -85,B 0,C 180,E1 -22649.922,E2 -22649.922} C_VEL
LIN {X 0,Y 192.204,Z 396.925,A -85,B 0,C 180,E1 -22651.692,E2 -22651.692} C_VEL
LIN {X 0,Y 191.25,Z 395.26,A -85,B 0,C 180,E1 -22652.507,E2 -22652.507} C_VEL
LIN {X 0,Y 188.853,Z 392.584,A -85,B 0,C 180,E1 -22654.44,E2 -22654.44} C_VEL
LIN {X 0,Y 187.607,Z 390.239,A -85,B 0,C 180,E1 -22655.665,E2 -22655.665} C_VEL
LIN {X 0,Y 184.97,Z 387.918,A -85,B 0,C 180,E1 -22657.963,E2 -22657.963} C_VEL
LIN {X 0,Y 183.621,Z 385.048,A -85,B 0,C 180,E1 -22659.558,E2 -22659.558} C_VEL
LIN {X 0,Y 183.386,Z 384.702,A -85,B 0,C 180,E1 -22659.823,E2 -22659.823} C_VEL
LIN {X 0,Y 180.395,Z 382.711,A -85,B 0,C 180,E1 -22663.011,E2 -22663.011} C_VEL
LIN {X 0,Y 178.969,Z 380.27,A -85,B 0,C 180,E1 -22665.066,E2 -22665.066} C_VEL
LIN {X 0,Y 178.653,Z 378.82,A -85,B 0,C 180,E1 -22665.839,E2 -22665.839} C_VEL
LIN {X 0,Y 178.976,Z 378.817,A -85,B 0,C 180,E1 -22670.963,E2 -22670.963} C_VEL
LIN {X 0,Y 179.153,Z 378.795,A -85,B 0,C 180,E1 -22677.752,E2 -22677.752} C_VEL
LIN {X 0,Y 179.371,Z 378.768,A -85,B 0,C 180,E1 -22680,E2 -22680} C_VEL
LIN {X 0,Y 178.876,Z 378.829,A -85,B 0,C 180,E1 -22684.507,E2 -22684.507} C_VEL
LIN {X 0,Y 179.02,Z 379.115,A -85,B 0,C 180,E1 -22689.034,E2 -22689.034} C_VEL
LIN {X 0,Y 178.977,Z 380.687,A -85,B 0,C 180,E1 -22694.279,E2 -22694.279} C_VEL
LIN {X 0,Y 180.101,Z 383.756,A -85,B 0,C 180,E1 -22696.07,E2 -22696.07} C_VEL
LIN {X 0,Y 182.869,Z 387.243,A -85,B 0,C 180,E1 -22699.268,E2 -22699.268} C_VEL
LIN {X 0,Y 184.165,Z 388.474,A -85,B 0,C 180,E1 -22700.524,E2 -22700.524} C_VEL
LIN {X 0,Y 185.626,Z 391.711,A -85,B 0,C 180,E1 -22702.101,E2 -22702.101} C_VEL
LIN {X 0,Y 188.612,Z 395.476,A -85,B 0,C 180,E1 -22704.71,E2 -22704.71} C_VEL
LIN {X 0,Y 190.541,Z 399.316,A -85,B 0,C 180,E1 -22706.418,E2 -22706.418} C_VEL
LIN {X 0,Y 192.273,Z 401.749,A -85,B 0,C 180,E1 -22707.777,E2 -22707.777} C_VEL
LIN {X 0,Y 194.477,Z 406.099,A -85,B 0,C 180,E1 -22709.571,E2 -22709.571} C_VEL
LIN {X 0,Y 195.627,Z 408.106,A -85,B 0,C 180,E1 -22710.436,E2 -22710.436} C_VEL
LIN {X 0,Y 198.435,Z 413.807,A -85,B 0,C 180,E1 -22712.621,E2 -22712.621} C_VEL
LIN {X 0,Y 201.644,Z 420.9,A -85,B 0,C 180,E1 -22715.105,E2 -22715.105} C_VEL
LIN {X 0,Y 205.232,Z 430.366,A -85,B 0,C 180,E1 -22718.053,E2 -22718.053} C_VEL
LIN {X 0,Y 206.667,Z 436.16,A -85,B 0,C 180,E1 -22719.614,E2 -22719.614} C_VEL
LIN {X 0,Y 208.092,Z 448.222,A -85,B 0,C 180,E1 -22722.49,E2 -22722.49} C_VEL
LIN {X 0,Y 208.291,Z 459.535,A -85,B 0,C 180,E1 -22725.118,E2 -22725.118} C_VEL
LIN {X 0,Y 207.522,Z 470.76,A -85,B 0,C 180,E1 -22727.822,E2 -22727.822} C_VEL
LIN {X 0,Y 206.76,Z 475.717,A -85,B 0,C 180,E1 -22729.036,E2 -22729.036} C_VEL
LIN {X 0,Y 201.185,Z 487.917,A -85,B 0,C 180,E1 -22731.681,E2 -22731.681} C_VEL
LIN {X 0,Y 196.261,Z 497.926,A -85,B 0,C 180,E1 -22734.417,E2 -22734.417} C_VEL
LIN {X 0,Y 191.559,Z 507.107,A -85,B 0,C 180,E1 -22737.547,E2 -22737.547} C_VEL
LIN {X 0,Y 186.968,Z 515.944,A -85,B 0,C 180,E1 -22741.364,E2 -22741.364} C_VEL
LIN {X 0,Y 183.206,Z 522.733,A -85,B 0,C 180,E1 -22745.042,E2 -22745.042} C_VEL
LIN {X 0,Y 179.938,Z 529.265,A -85,B 0,C 180,E1 -22749.617,E2 -22749.617} C_VEL
LIN {X 0,Y 177.838,Z 533.911,A -85,B 0,C 180,E1 -22753.942,E2 -22753.942} C_VEL
LIN {X 0,Y 176.509,Z 537.505,A -85,B 0,C 180,E1 -22758.518,E2 -22758.518} C_VEL
LIN {X 0,Y 176.108,Z 539.89,A -85,B 0,C 180,E1 -22763.125,E2 -22763.125} C_VEL
LIN {X 0,Y 176.145,Z 540.751,A -85,B 0,C 180,E1 -22765.921,E2 -22765.921} C_VEL
LIN {X 0,Y 176.33,Z 541.264,A -85,B 0,C 180,E1 -22770.001,E2 -22770.001} C_VEL
LIN {X 0,Y 176.219,Z 541.182,A -85,B 0,C 180,E1 -22771.105,E2 -22771.105} C_VEL
LIN {X 0,Y 175.435,Z 540.939,A -85,B 0,C 180,E1 -22773.008,E2 -22773.008} C_VEL
LIN {X 0,Y 172.494,Z 540.01,A -85,B 0,C 180,E1 -22776.113,E2 -22776.113} C_VEL
LIN {X 0,Y 170.169,Z 538.93,A -85,B 0,C 180,E1 -22778.653,E2 -22778.653} C_VEL
LIN {X 0,Y 169.341,Z 537.744,A -85,B 0,C 180,E1 -22780.951,E2 -22780.951} C_VEL
LIN {X 0,Y 169.375,Z 537.495,A -85,B 0,C 180,E1 -22781.282,E2 -22781.282} C_VEL
LIN {X 0,Y 170.067,Z 535.458,A -85,B 0,C 180,E1 -22784.357,E2 -22784.357} C_VEL
LIN {X 0,Y 172.036,Z 531.219,A -85,B 0,C 180,E1 -22789.077,E2 -22789.077} C_VEL
LIN {X 0,Y 174.899,Z 525.622,A -85,B 0,C 180,E1 -22793.694,E2 -22793.694} C_VEL
LIN {X 0,Y 178.845,Z 518.531,A -85,B 0,C 180,E1 -22798.137,E2 -22798.137} C_VEL
LIN {X 0,Y 183.197,Z 510.97,A -85,B 0,C 180,E1 -22801.837,E2 -22801.837} C_VEL
LIN {X 0,Y 188.109,Z 501.86,A -85,B 0,C 180,E1 -22805.388,E2 -22805.388} C_VEL
LIN {X 0,Y 193.884,Z 490.936,A -85,B 0,C 180,E1 -22808.704,E2 -22808.704} C_VEL
LIN {X 0,Y 198.425,Z 481.669,A -85,B 0,C 180,E1 -22810.94,E2 -22810.94} C_VEL
LIN {X 0,Y 200.765,Z 476.491,A -85,B 0,C 180,E1 -22812.036,E2 -22812.036} C_VEL
LIN {X 0,Y 202.042,Z 467.034,A -85,B 0,C 180,E1 -22814.484,E2 -22814.484} C_VEL
LIN {X 0,Y 202.534,Z 457.074,A -85,B 0,C 180,E1 -22816.951,E2 -22816.951} C_VEL
LIN {X 0,Y 202.201,Z 446.004,A -85,B 0,C 180,E1 -22819.69,E2 -22819.69} C_VEL
LIN {X 0,Y 201.044,Z 437.236,A -85,B 0,C 180,E1 -22821.958,E2 -22821.958} C_VEL
LIN {X 0,Y 199.208,Z 430.956,A -85,B 0,C 180,E1 -22823.903,E2 -22823.903} C_VEL
LIN {X 0,Y 196.001,Z 422.333,A -85,B 0,C 180,E1 -22826.851,E2 -22826.851} C_VEL
LIN {X 0,Y 193.659,Z 417.096,A -85,B 0,C 180,E1 -22828.86,E2 -22828.86} C_VEL
LIN {X 0,Y 191.25,Z 412.044,A -85,B 0,C 180,E1 -22830.957,E2 -22830.957} C_VEL
LIN {X 0,Y 189.072,Z 407.373,A -85,B 0,C 180,E1 -22832.988,E2 -22832.988} C_VEL
LIN {X 0,Y 186.479,Z 403.114,A -85,B 0,C 180,E1 -22835.285,E2 -22835.285} C_VEL
LIN {X 0,Y 185.575,Z 401.106,A -85,B 0,C 180,E1 -22836.236,E2 -22836.236} C_VEL
LIN {X 0,Y 183.013,Z 397.491,A -85,B 0,C 180,E1 -22838.752,E2 -22838.752} C_VEL
LIN {X 0,Y 181.658,Z 394.47,A -85,B 0,C 180,E1 -22840.37,E2 -22840.37} C_VEL
LIN {X 0,Y 178.802,Z 391.07,A -85,B 0,C 180,E1 -22843.737,E2 -22843.737} C_VEL
LIN {X 0,Y 177.415,Z 387.573,A -85,B 0,C 180,E1 -22846.031,E2 -22846.031} C_VEL
LIN {X 0,Y 173.843,Z 383.769,A -85,B 0,C 180,E1 -22853.034,E2 -22853.034} C_VEL
LIN {X 0,Y 172.76,Z 381.306,A -85,B 0,C 180,E1 -22860,E2 -22860} C_VEL
LIN {X 0,Y 177.083,Z 385.944,A -85,B 0,C 180,E1 -22874.142,E2 -22874.142} C_VEL
LIN {X 0,Y 178.169,Z 388.743,A -85,B 0,C 180,E1 -22876.176,E2 -22876.176} C_VEL
LIN {X 0,Y 180.717,Z 391.124,A -85,B 0,C 180,E1 -22879.303,E2 -22879.303} C_VEL
LIN {X 0,Y 181.477,Z 391.685,A -85,B 0,C 180,E1 -22880.103,E2 -22880.103} C_VEL
LIN {X 0,Y 182.956,Z 394.689,A -85,B 0,C 180,E1 -22881.996,E2 -22881.996} C_VEL
LIN {X 0,Y 185.419,Z 397.227,A -85,B 0,C 180,E1 -22884.343,E2 -22884.343} C_VEL
LIN {X 0,Y 187.486,Z 400.64,A -85,B 0,C 180,E1 -22886.403,E2 -22886.403} C_VEL
LIN {X 0,Y 188.743,Z 402.13,A -85,B 0,C 180,E1 -22887.481,E2 -22887.481} C_VEL
LIN {X 0,Y 190.078,Z 404.575,A -85,B 0,C 180,E1 -22888.729,E2 -22888.729} C_VEL
LIN {X 0,Y 191.885,Z 407.158,A -85,B 0,C 180,E1 -22890.239,E2 -22890.239} C_VEL
LIN {X 0,Y 196.061,Z 414.403,A -85,B 0,C 180,E1 -22893.753,E2 -22893.753} C_VEL
LIN {X 0,Y 199.609,Z 421.545,A -85,B 0,C 180,E1 -22896.766,E2 -22896.766} C_VEL
LIN {X 0,Y 202.407,Z 428.328,A -85,B 0,C 180,E1 -22899.323,E2 -22899.323} C_VEL
LIN {X 0,Y 204.216,Z 434.966,A -85,B 0,C 180,E1 -22901.49,E2 -22901.49} C_VEL
LIN {X 0,Y 205.729,Z 443.768,A -85,B 0,C 180,E1 -22904.159,E2 -22904.159} C_VEL
LIN {X 0,Y 206.483,Z 453.752,A -85,B 0,C 180,E1 -22907.098,E2 -22907.098} C_VEL
LIN {X 0,Y 202.355,Z 463.709,A -85,B 0,C 180,E1 -22909.038,E2 -22909.038} C_VEL
LIN {X 0,Y 196.694,Z 475.483,A -85,B 0,C 180,E1 -22911.821,E2 -22911.821} C_VEL
LIN {X 0,Y 191.769,Z 485.121,A -85,B 0,C 180,E1 -22914.744,E2 -22914.744} C_VEL
LIN {X 0,Y 186.633,Z 494.264,A -85,B 0,C 180,E1 -22918.183,E2 -22918.183} C_VEL
LIN {X 0,Y 182.73,Z 500.862,A -85,B 0,C 180,E1 -22921.264,E2 -22921.264} C_VEL
LIN {X 0,Y 178.31,Z 508.145,A -85,B 0,C 180,E1 -22925.552,E2 -22925.552} C_VEL
LIN {X 0,Y 174.834,Z 513.91,A -85,B 0,C 180,E1 -22930.02,E2 -22930.02} C_VEL
LIN {X 0,Y 172.815,Z 517.317,A -85,B 0,C 180,E1 -22933.46,E2 -22933.46} C_VEL
LIN {X 0,Y 170.881,Z 520.758,A -85,B 0,C 180,E1 -22938.132,E2 -22938.132} C_VEL
LIN {X 0,Y 169.792,Z 523.022,A -85,B 0,C 180,E1 -22942.866,E2 -22942.866} C_VEL
LIN {X 0,Y 169.376,Z 524.168,A -85,B 0,C 180,E1 -22947.621,E2 -22947.621} C_VEL
LIN {X 0,Y 169.37,Z 524.179,A -85,B 0,C 180,E1 -22952.377,E2 -22952.377} C_VEL
LIN {X 0,Y 169.777,Z 523.078,A -85,B 0,C 180,E1 -22957.133,E2 -22957.133} C_VEL
LIN {X 0,Y 170.873,Z 520.858,A -85,B 0,C 180,E1 -22961.867,E2 -22961.867} C_VEL
LIN {X 0,Y 172.768,Z 517.457,A -85,B 0,C 180,E1 -22966.543,E2 -22966.543} C_VEL
LIN {X 0,Y 175.624,Z 512.786,A -85,B 0,C 180,E1 -22971.109,E2 -22971.109} C_VEL
LIN {X 0,Y 179.256,Z 506.643,A -85,B 0,C 180,E1 -22975.61,E2 -22975.61} C_VEL
LIN {X 0,Y 183.921,Z 499.084,A -85,B 0,C 180,E1 -22979.785,E2 -22979.785} C_VEL
LIN {X 0,Y 188.67,Z 490.925,A -85,B 0,C 180,E1 -22983.328,E2 -22983.328} C_VEL
LIN {X 0,Y 194.063,Z 481.082,A -85,B 0,C 180,E1 -22986.693,E2 -22986.693} C_VEL
LIN {X 0,Y 199.009,Z 470.992,A -85,B 0,C 180,E1 -22989.469,E2 -22989.469} C_VEL
LIN {X 0,Y 204.621,Z 458.945,A -85,B 0,C 180,E1 -22992.047,E2 -22992.047} C_VEL
LIN {X 0,Y 206.395,Z 454.345,A -85,B 0,C 180,E1 -22992.923,E2 -22992.923} C_VEL
